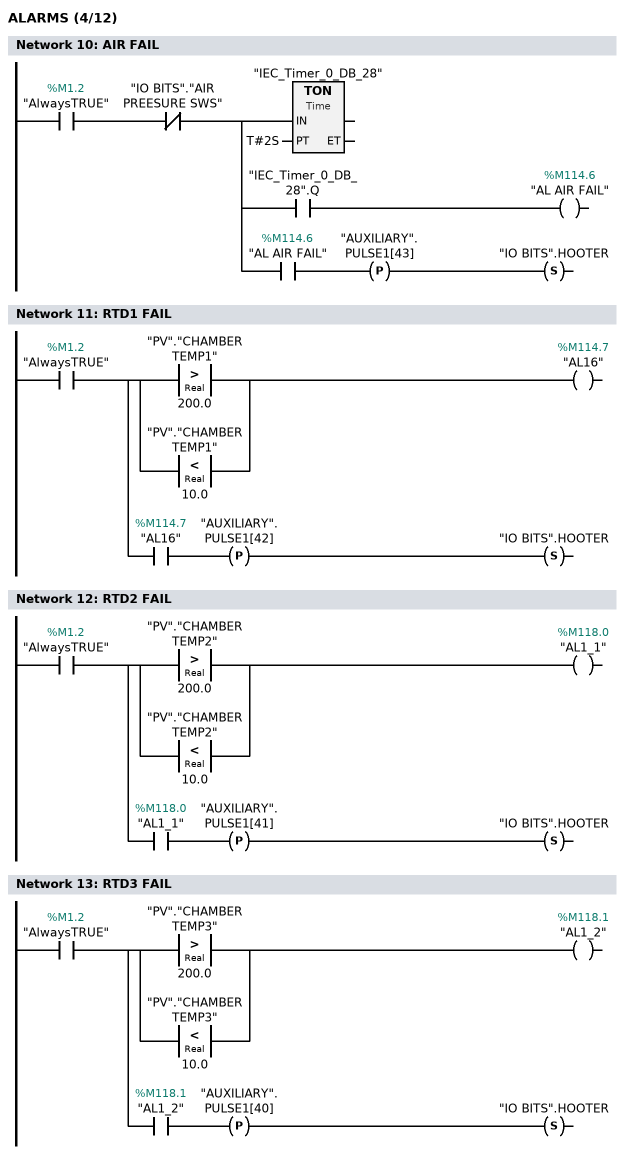
   RUNG wire#powerrail
      Contact( "AlwaysTRUE" )
      I_Contact( "IO BITS"."AIR PREESURE SWS" )
      wire#w1
      { S7_Templates := "time_type := Time" } "IEC_Timer_0_DB_28".TON(pt := T#2S, et =>)
   END_RUNG
   RUNG wire#w1
      Contact( "IEC_Timer_0_DB_28".Q )
      Coil( "AL AIR FAIL" )
   END_RUNG
   RUNG wire#w1
      Contact( "AL AIR FAIL" )
      P_Trig( "AUXILIARY".PULSE1[43] )
      S_Coil( "IO BITS".HOOTER )
   END_RUNG
   // the same network as SCL:
   #_w1 := "AlwaysTRUE" AND NOT "IO BITS"."AIR PREESURE SWS";
   "IEC_Timer_0_DB_28".TON(IN := #_w1, PT := T#2S);
   "AL AIR FAIL" := #_w1 AND "IEC_Timer_0_DB_28".Q;
   #_w2 := #_w1 AND "AL AIR FAIL";
   #_w3 := #_w2 AND NOT "AUXILIARY".PULSE1[43];   // rising edge
   "AUXILIARY".PULSE1[43] := #_w2;
   IF #_w3 THEN "IO BITS".HOOTER := TRUE; END_IF;
END_REGION

REGION Network 11: RTD1 FAIL
   RUNG wire#powerrail
      Contact( "AlwaysTRUE" )
      wire#w1
      { S7_Templates := "SrcType := Real" } GT_Contact(in1 := "PV"."CHAMBER TEMP1", in2 := 200.0)
      wire#w2
      Coil( "AL16" )
   END_RUNG
   RUNG wire#w1
      { S7_Templates := "SrcType := Real" } LT_Contact(in1 := "PV"."CHAMBER TEMP1", in2 := 10.0)
   END_RUNG wire#w2
   RUNG wire#w1
      Contact( "AL16" )
      P_Trig( "AUXILIARY".PULSE1[42] )
      S_Coil( "IO BITS".HOOTER )
   END_RUNG
   // the same network as SCL:
   "AL16" := "AlwaysTRUE" AND (("PV"."CHAMBER TEMP1" > 200.0) OR ("PV"."CHAMBER TEMP1" < 10.0));
   #_w1 := "AlwaysTRUE" AND "AL16";
   #_w2 := #_w1 AND NOT "AUXILIARY".PULSE1[42];   // rising edge
   "AUXILIARY".PULSE1[42] := #_w1;
   IF #_w2 THEN "IO BITS".HOOTER := TRUE; END_IF;
END_REGION

REGION Network 12: RTD2 FAIL
   RUNG wire#powerrail
      Contact( "AlwaysTRUE" )
      wire#w1
      { S7_Templates := "SrcType := Real" } GT_Contact(in1 := "PV"."CHAMBER TEMP2", in2 := 200.0)
      wire#w2
      Coil( "AL1_1" )
   END_RUNG
   RUNG wire#w1
      { S7_Templates := "SrcType := Real" } LT_Contact(in1 := "PV"."CHAMBER TEMP2", in2 := 10.0)
   END_RUNG wire#w2
   RUNG wire#w1
      Contact( "AL1_1" )
      P_Trig( "AUXILIARY".PULSE1[41] )
      S_Coil( "IO BITS".HOOTER )
   END_RUNG
   // the same network as SCL:
   "AL1_1" := "AlwaysTRUE" AND (("PV"."CHAMBER TEMP2" > 200.0) OR ("PV"."CHAMBER TEMP2" < 10.0));
   #_w1 := "AlwaysTRUE" AND "AL1_1";
   #_w2 := #_w1 AND NOT "AUXILIARY".PULSE1[41];   // rising edge
   "AUXILIARY".PULSE1[41] := #_w1;
   IF #_w2 THEN "IO BITS".HOOTER := TRUE; END_IF;
END_REGION

REGION Network 13: RTD3 FAIL
   RUNG wire#powerrail
      Contact( "AlwaysTRUE" )
      wire#w1
      { S7_Templates := "SrcType := Real" } GT_Contact(in1 := "PV"."CHAMBER TEMP3", in2 := 200.0)
      wire#w2
      Coil( "AL1_2" )
   END_RUNG
   RUNG wire#w1
      { S7_Templates := "SrcType := Real" } LT_Contact(in1 := "PV"."CHAMBER TEMP3", in2 := 10.0)
   END_RUNG wire#w2
   RUNG wire#w1
      Contact( "AL1_2" )
      P_Trig( "AUXILIARY".PULSE1[40] )
      S_Coil( "IO BITS".HOOTER )
   END_RUNG
   // the same network as SCL:
   "AL1_2" := "AlwaysTRUE" AND (("PV"."CHAMBER TEMP3" > 200.0) OR ("PV"."CHAMBER TEMP3" < 10.0));
   #_w1 := "AlwaysTRUE" AND "AL1_2";
   #_w2 := #_w1 AND NOT "AUXILIARY".PULSE1[40];   // rising edge
   "AUXILIARY".PULSE1[40] := #_w1;
   IF #_w2 THEN "IO BITS".HOOTER := TRUE; END_IF;
END_REGION

REGION Network 14: RTD4 FAIL
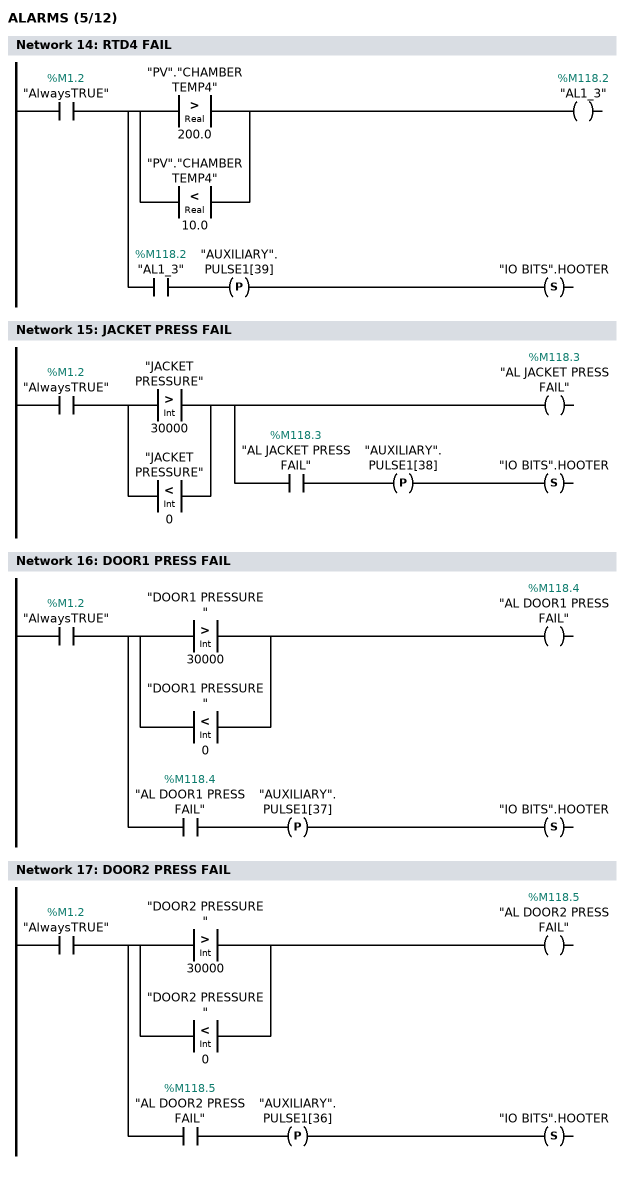
   RUNG wire#powerrail
      Contact( "AlwaysTRUE" )
      wire#w1
      { S7_Templates := "SrcType := Real" } GT_Contact(in1 := "PV"."CHAMBER TEMP4", in2 := 200.0)
      wire#w2
      Coil( "AL1_3" )
   END_RUNG
   RUNG wire#w1
      { S7_Templates := "SrcType := Real" } LT_Contact(in1 := "PV"."CHAMBER TEMP4", in2 := 10.0)
   END_RUNG wire#w2
   RUNG wire#w1
      Contact( "AL1_3" )
      P_Trig( "AUXILIARY".PULSE1[39] )
      S_Coil( "IO BITS".HOOTER )
   END_RUNG
   // the same network as SCL:
   "AL1_3" := "AlwaysTRUE" AND (("PV"."CHAMBER TEMP4" > 200.0) OR ("PV"."CHAMBER TEMP4" < 10.0));
   #_w1 := "AlwaysTRUE" AND "AL1_3";
   #_w2 := #_w1 AND NOT "AUXILIARY".PULSE1[39];   // rising edge
   "AUXILIARY".PULSE1[39] := #_w1;
   IF #_w2 THEN "IO BITS".HOOTER := TRUE; END_IF;
END_REGION

REGION Network 15: JACKET PRESS FAIL
   RUNG wire#powerrail
      Contact( "AlwaysTRUE" )
      wire#w1
      { S7_Templates := "SrcType := Int" } GT_Contact(in1 := "JACKET PRESSURE", in2 := 30000)
      wire#w2
      Coil( "AL JACKET PRESS FAIL" )
   END_RUNG
   RUNG wire#w1
      { S7_Templates := "SrcType := Int" } LT_Contact(in1 := "JACKET PRESSURE", in2 := 0)
   END_RUNG wire#w2
   RUNG wire#w2
      Contact( "AL JACKET PRESS FAIL" )
      P_Trig( "AUXILIARY".PULSE1[38] )
      S_Coil( "IO BITS".HOOTER )
   END_RUNG
   // the same network as SCL:
   "AL JACKET PRESS FAIL" := "AlwaysTRUE" AND (("JACKET PRESSURE" > 30000) OR ("JACKET PRESSURE" < 0));
   #_w1 := "AL JACKET PRESS FAIL" AND "AL JACKET PRESS FAIL";
   #_w2 := #_w1 AND NOT "AUXILIARY".PULSE1[38];   // rising edge
   "AUXILIARY".PULSE1[38] := #_w1;
   IF #_w2 THEN "IO BITS".HOOTER := TRUE; END_IF;
END_REGION

REGION Network 16: DOOR1 PRESS FAIL
   RUNG wire#powerrail
      Contact( "AlwaysTRUE" )
      wire#w1
      { S7_Templates := "SrcType := Int" } GT_Contact(in1 := "DOOR1 PRESSURE", in2 := 30000)
      wire#w2
      Coil( "AL DOOR1 PRESS FAIL" )
   END_RUNG
   RUNG wire#w1
      { S7_Templates := "SrcType := Int" } LT_Contact(in1 := "DOOR1 PRESSURE", in2 := 0)
   END_RUNG wire#w2
   RUNG wire#w1
      Contact( "AL DOOR1 PRESS FAIL" )
      P_Trig( "AUXILIARY".PULSE1[37] )
      S_Coil( "IO BITS".HOOTER )
   END_RUNG
   // the same network as SCL:
   "AL DOOR1 PRESS FAIL" := "AlwaysTRUE" AND (("DOOR1 PRESSURE" > 30000) OR ("DOOR1 PRESSURE" < 0));
   #_w1 := "AlwaysTRUE" AND "AL DOOR1 PRESS FAIL";
   #_w2 := #_w1 AND NOT "AUXILIARY".PULSE1[37];   // rising edge
   "AUXILIARY".PULSE1[37] := #_w1;
   IF #_w2 THEN "IO BITS".HOOTER := TRUE; END_IF;
END_REGION

REGION Network 17: DOOR2 PRESS FAIL
   RUNG wire#powerrail
      Contact( "AlwaysTRUE" )
      wire#w1
      { S7_Templates := "SrcType := Int" } GT_Contact(in1 := "DOOR2 PRESSURE", in2 := 30000)
      wire#w2
      Coil( "AL DOOR2 PRESS FAIL" )
   END_RUNG
   RUNG wire#w1
      { S7_Templates := "SrcType := Int" } LT_Contact(in1 := "DOOR2 PRESSURE", in2 := 0)
   END_RUNG wire#w2
   RUNG wire#w1
      Contact( "AL DOOR2 PRESS FAIL" )
      P_Trig( "AUXILIARY".PULSE1[36] )
      S_Coil( "IO BITS".HOOTER )
   END_RUNG
   // the same network as SCL:
   "AL DOOR2 PRESS FAIL" := "AlwaysTRUE" AND (("DOOR2 PRESSURE" > 30000) OR ("DOOR2 PRESSURE" < 0));
   #_w1 := "AlwaysTRUE" AND "AL DOOR2 PRESS FAIL";
   #_w2 := #_w1 AND NOT "AUXILIARY".PULSE1[36];   // rising edge
   "AUXILIARY".PULSE1[36] := #_w1;
   IF #_w2 THEN "IO BITS".HOOTER := TRUE; END_IF;
END_REGION

REGION Network 18: chamber press fail
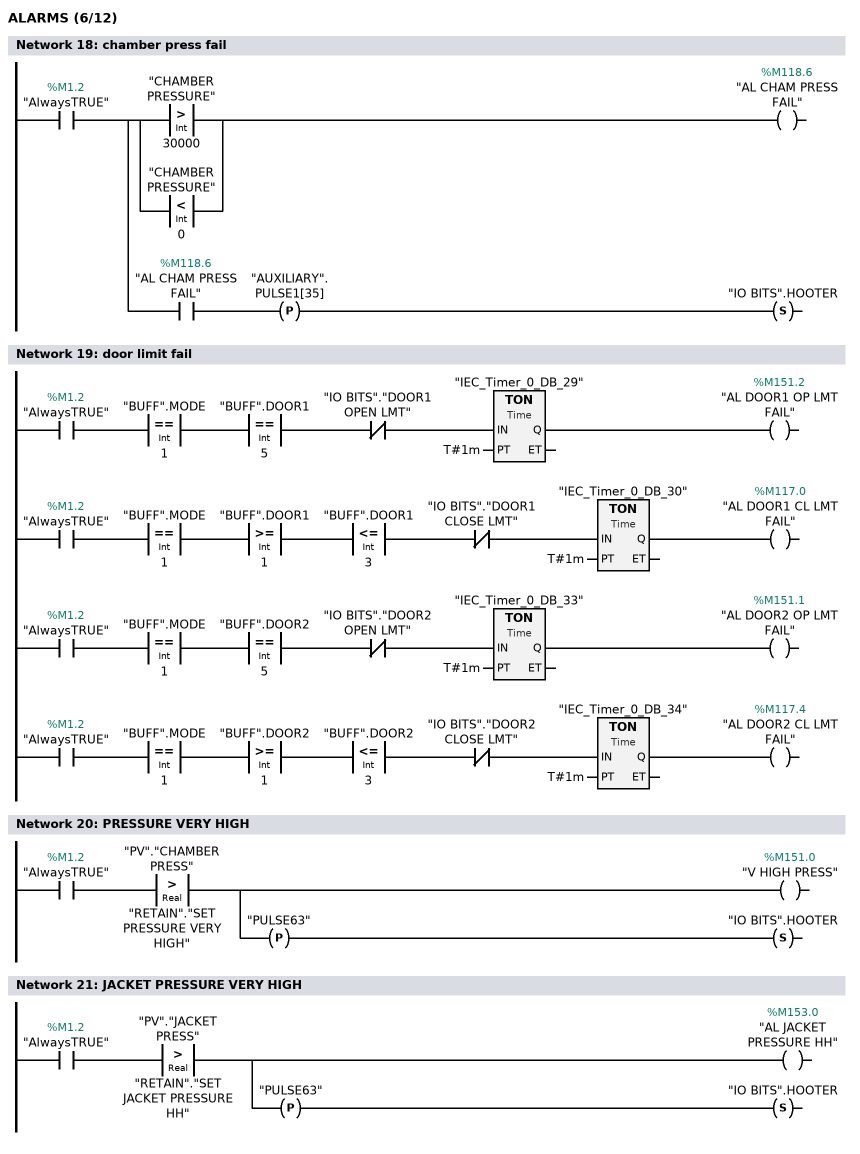
   RUNG wire#powerrail
      Contact( "AlwaysTRUE" )
      wire#w1
      { S7_Templates := "SrcType := Int" } GT_Contact(in1 := "CHAMBER PRESSURE", in2 := 30000)
      wire#w2
      Coil( "AL CHAM PRESS FAIL" )
   END_RUNG
   RUNG wire#w1
      { S7_Templates := "SrcType := Int" } LT_Contact(in1 := "CHAMBER PRESSURE", in2 := 0)
   END_RUNG wire#w2
   RUNG wire#w1
      Contact( "AL CHAM PRESS FAIL" )
      P_Trig( "AUXILIARY".PULSE1[35] )
      S_Coil( "IO BITS".HOOTER )
   END_RUNG
   // the same network as SCL:
   "AL CHAM PRESS FAIL" := "AlwaysTRUE" AND (("CHAMBER PRESSURE" > 30000) OR ("CHAMBER PRESSURE" < 0));
   #_w1 := "AlwaysTRUE" AND "AL CHAM PRESS FAIL";
   #_w2 := #_w1 AND NOT "AUXILIARY".PULSE1[35];   // rising edge
   "AUXILIARY".PULSE1[35] := #_w1;
   IF #_w2 THEN "IO BITS".HOOTER := TRUE; END_IF;
END_REGION

REGION Network 19: door limit fail
   RUNG wire#powerrail
      Contact( "AlwaysTRUE" )
      { S7_Templates := "SrcType := Int" } EQ_Contact(in1 := "BUFF".MODE, in2 := 1)
      { S7_Templates := "SrcType := Int" } EQ_Contact(in1 := "BUFF".DOOR1, in2 := 5)
      I_Contact( "IO BITS"."DOOR1 OPEN LMT" )
      { S7_Templates := "time_type := Time" } "IEC_Timer_0_DB_29".TON(pt := T#1m, et =>)
      Coil( "AL DOOR1 OP LMT FAIL" )
   END_RUNG
   RUNG wire#powerrail
      Contact( "AlwaysTRUE" )
      { S7_Templates := "SrcType := Int" } EQ_Contact(in1 := "BUFF".MODE, in2 := 1)
      { S7_Templates := "SrcType := Int" } GE_Contact(in1 := "BUFF".DOOR1, in2 := 1)
      { S7_Templates := "SrcType := Int" } LE_Contact(in1 := "BUFF".DOOR1, in2 := 3)
      I_Contact( "IO BITS"."DOOR1 CLOSE LMT" )
      { S7_Templates := "time_type := Time" } "IEC_Timer_0_DB_30".TON(pt := T#1m, et =>)
      Coil( "AL DOOR1 CL LMT FAIL" )
   END_RUNG
   RUNG wire#powerrail
      Contact( "AlwaysTRUE" )
      { S7_Templates := "SrcType := Int" } EQ_Contact(in1 := "BUFF".MODE, in2 := 1)
      { S7_Templates := "SrcType := Int" } EQ_Contact(in1 := "BUFF".DOOR2, in2 := 5)
      I_Contact( "IO BITS"."DOOR2 OPEN LMT" )
      { S7_Templates := "time_type := Time" } "IEC_Timer_0_DB_33".TON(pt := T#1m, et =>)
      Coil( "AL DOOR2 OP LMT FAIL" )
   END_RUNG
   RUNG wire#powerrail
      Contact( "AlwaysTRUE" )
      { S7_Templates := "SrcType := Int" } EQ_Contact(in1 := "BUFF".MODE, in2 := 1)
      { S7_Templates := "SrcType := Int" } GE_Contact(in1 := "BUFF".DOOR2, in2 := 1)
      { S7_Templates := "SrcType := Int" } LE_Contact(in1 := "BUFF".DOOR2, in2 := 3)
      I_Contact( "IO BITS"."DOOR2 CLOSE LMT" )
      { S7_Templates := "time_type := Time" } "IEC_Timer_0_DB_34".TON(pt := T#1m, et =>)
      Coil( "AL DOOR2 CL LMT FAIL" )
   END_RUNG
   // the same network as SCL:
   "IEC_Timer_0_DB_29".TON(IN := "AlwaysTRUE" AND ("BUFF".MODE = 1) AND ("BUFF".DOOR1 = 5) AND NOT "IO BITS"."DOOR1 OPEN LMT",
                           PT := T#1m);
   "AL DOOR1 OP LMT FAIL" := "IEC_Timer_0_DB_29".Q;
   "IEC_Timer_0_DB_30".TON(IN := "AlwaysTRUE" AND ("BUFF".MODE = 1) AND ("BUFF".DOOR1 >= 1) AND ("BUFF".DOOR1 <= 3) AND NOT "IO BITS"."DOOR1 CLOSE LMT",
                           PT := T#1m);
   "AL DOOR1 CL LMT FAIL" := "IEC_Timer_0_DB_30".Q;
   "IEC_Timer_0_DB_33".TON(IN := "AlwaysTRUE" AND ("BUFF".MODE = 1) AND ("BUFF".DOOR2 = 5) AND NOT "IO BITS"."DOOR2 OPEN LMT",
                           PT := T#1m);
   "AL DOOR2 OP LMT FAIL" := "IEC_Timer_0_DB_33".Q;
   "IEC_Timer_0_DB_34".TON(IN := "AlwaysTRUE" AND ("BUFF".MODE = 1) AND ("BUFF".DOOR2 >= 1) AND ("BUFF".DOOR2 <= 3) AND NOT "IO BITS"."DOOR2 CLOSE LMT",
                           PT := T#1m);
   "AL DOOR2 CL LMT FAIL" := "IEC_Timer_0_DB_34".Q;
END_REGION

REGION Network 20: PRESSURE VERY HIGH
   RUNG wire#powerrail
      Contact( "AlwaysTRUE" )
      { S7_Templates := "SrcType := Real" } GT_Contact(in1 := "PV"."CHAMBER PRESS", in2 := "RETAIN"."SET PRESSURE VERY HIGH")
      wire#w1
      Coil( "V HIGH PRESS" )
   END_RUNG
   RUNG wire#w1
      P_Trig( "PULSE63" )
      S_Coil( "IO BITS".HOOTER )
   END_RUNG
   // the same network as SCL:
   "V HIGH PRESS" := "AlwaysTRUE" AND ("PV"."CHAMBER PRESS" > "RETAIN"."SET PRESSURE VERY HIGH");
   #_w1 := "V HIGH PRESS" AND NOT "PULSE63";   // rising edge
   "PULSE63" := "V HIGH PRESS";
   IF #_w1 THEN "IO BITS".HOOTER := TRUE; END_IF;
END_REGION

REGION Network 21: JACKET PRESSURE VERY HIGH
   RUNG wire#powerrail
      Contact( "AlwaysTRUE" )
      { S7_Templates := "SrcType := Real" } GT_Contact(in1 := "PV"."JACKET PRESS", in2 := "RETAIN"."SET JACKET PRESSURE HH")
      wire#w1
      Coil( "AL JACKET PRESSURE HH" )
   END_RUNG
   RUNG wire#w1
      P_Trig( "PULSE63" )
      S_Coil( "IO BITS".HOOTER )
   END_RUNG
   // the same network as SCL:
   "AL JACKET PRESSURE HH" := "AlwaysTRUE" AND ("PV"."JACKET PRESS" > "RETAIN"."SET JACKET PRESSURE HH");
   #_w1 := "AL JACKET PRESSURE HH" AND NOT "PULSE63";   // rising edge
   "PULSE63" := "AL JACKET PRESSURE HH";
   IF #_w1 THEN "IO BITS".HOOTER := TRUE; END_IF;
END_REGION

REGION Network 22: TEMPERATURE OVERSHOOT
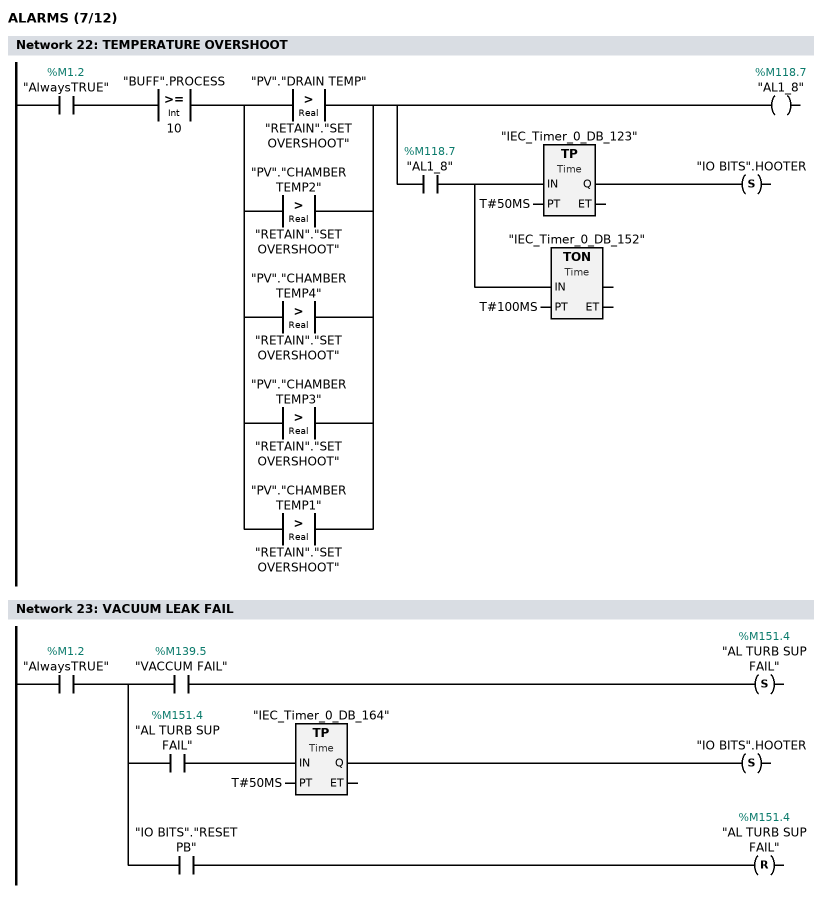
   RUNG wire#powerrail
      Contact( "AlwaysTRUE" )
      { S7_Templates := "SrcType := Int" } GE_Contact(in1 := "BUFF".PROCESS, in2 := 10)
      wire#w1
      { S7_Templates := "SrcType := Real" } GT_Contact(in1 := "PV"."DRAIN TEMP", in2 := "RETAIN"."SET OVERSHOOT")
      wire#w2
      Coil( "AL1_8" )
   END_RUNG
   RUNG wire#w1
      { S7_Templates := "SrcType := Real" } GT_Contact(in1 := "PV"."CHAMBER TEMP2", in2 := "RETAIN"."SET OVERSHOOT")
   END_RUNG wire#w2
   RUNG wire#w1
      { S7_Templates := "SrcType := Real" } GT_Contact(in1 := "PV"."CHAMBER TEMP4", in2 := "RETAIN"."SET OVERSHOOT")
   END_RUNG wire#w2
   RUNG wire#w1
      { S7_Templates := "SrcType := Real" } GT_Contact(in1 := "PV"."CHAMBER TEMP3", in2 := "RETAIN"."SET OVERSHOOT")
   END_RUNG wire#w2
   RUNG wire#w1
      { S7_Templates := "SrcType := Real" } GT_Contact(in1 := "PV"."CHAMBER TEMP1", in2 := "RETAIN"."SET OVERSHOOT")
   END_RUNG wire#w2
   RUNG wire#w2
      Contact( "AL1_8" )
      wire#w3
      { S7_Templates := "time_type := Time" } "IEC_Timer_0_DB_123".TP(pt := T#50MS, et =>)
      S_Coil( "IO BITS".HOOTER )
   END_RUNG
   RUNG wire#w3
      { S7_Templates := "time_type := Time" } "IEC_Timer_0_DB_152".TON(pt := T#100MS, et =>)
   END_RUNG
   // the same network as SCL:
   "AL1_8" := "AlwaysTRUE" AND ("BUFF".PROCESS >= 10) AND (("PV"."DRAIN TEMP" > "RETAIN"."SET OVERSHOOT") OR ("PV"."CHAMBER TEMP2" > "RETAIN"."SET OVERSHOOT") OR ("PV"."CHAMBER TEMP4" > "RETAIN"."SET OVERSHOOT") OR ("PV"."CHAMBER TEMP3" > "RETAIN"."SET OVERSHOOT") OR ("PV"."CHAMBER TEMP1" > "RETAIN"."SET OVERSHOOT"));
   #_w1 := "AL1_8" AND "AL1_8";
   "IEC_Timer_0_DB_123".TP(IN := #_w1, PT := T#50MS);
   IF "IEC_Timer_0_DB_123".Q THEN "IO BITS".HOOTER := TRUE; END_IF;
   "IEC_Timer_0_DB_152".TON(IN := #_w1, PT := T#100MS);
END_REGION

REGION Network 23: VACUUM LEAK FAIL
   RUNG wire#powerrail
      Contact( "AlwaysTRUE" )
      wire#w1
      Contact( "VACCUM FAIL" )
      S_Coil( "AL TURB SUP FAIL" )
   END_RUNG
   RUNG wire#w1
      Contact( "AL TURB SUP FAIL" )
      { S7_Templates := "time_type := Time" } "IEC_Timer_0_DB_164".TP(pt := T#50MS, et =>)
      S_Coil( "IO BITS".HOOTER )
   END_RUNG
   RUNG wire#w1
      Contact( "IO BITS"."RESET PB" )
      R_Coil( "AL TURB SUP FAIL" )
   END_RUNG
   // the same network as SCL:
   IF "AlwaysTRUE" AND "VACCUM FAIL" THEN "AL TURB SUP FAIL" := TRUE; END_IF;
   "IEC_Timer_0_DB_164".TP(IN := "AlwaysTRUE" AND "AL TURB SUP FAIL", PT := T#50MS);
   IF "IEC_Timer_0_DB_164".Q THEN "IO BITS".HOOTER := TRUE; END_IF;
   IF "AlwaysTRUE" AND "IO BITS"."RESET PB" THEN "AL TURB SUP FAIL" := FALSE; END_IF;
END_REGION

REGION Network 24: vacuum break fail
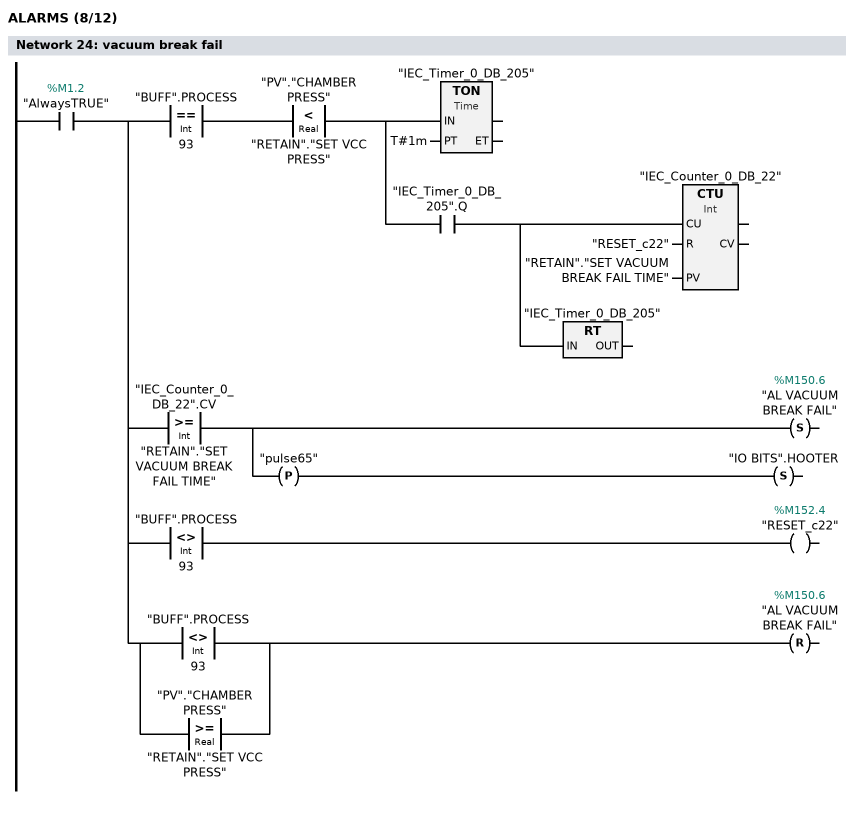
   RUNG wire#powerrail
      Contact( "AlwaysTRUE" )
      wire#w1
      { S7_Templates := "SrcType := Int" } EQ_Contact(in1 := "BUFF".PROCESS, in2 := 93)
      { S7_Templates := "SrcType := Real" } LT_Contact(in1 := "PV"."CHAMBER PRESS", in2 := "RETAIN"."SET VCC PRESS")
      wire#w2
      { S7_Templates := "time_type := Time" } "IEC_Timer_0_DB_205".TON(pt := T#1m, et =>)
   END_RUNG
   RUNG wire#w2
      Contact( "IEC_Timer_0_DB_205".Q )
      wire#w3
      { S7_Templates := "value_type := Int" } "IEC_Counter_0_DB_22".CTU(r := "RESET_c22", pv := "RETAIN"."SET VACUUM BREAK FAIL TIME", cv =>)
   END_RUNG
   RUNG wire#w3
      RT_Coil( "IEC_Timer_0_DB_205" )
   END_RUNG
   RUNG wire#w1
      { S7_Templates := "SrcType := Int" } GE_Contact(in1 := "IEC_Counter_0_DB_22".CV, in2 := "RETAIN"."SET VACUUM BREAK FAIL TIME")
      wire#w4
      S_Coil( "AL VACUUM BREAK FAIL" )
   END_RUNG
   RUNG wire#w4
      P_Trig( "pulse65" )
      S_Coil( "IO BITS".HOOTER )
   END_RUNG
   RUNG wire#w1
      { S7_Templates := "SrcType := Int" } NE_Contact(in1 := "BUFF".PROCESS, in2 := 93)
      Coil( "RESET_c22" )
   END_RUNG
   RUNG wire#w1
      { S7_Templates := "SrcType := Int" } NE_Contact(in1 := "BUFF".PROCESS, in2 := 93)
      wire#w5
      R_Coil( "AL VACUUM BREAK FAIL" )
   END_RUNG
   RUNG wire#w1
      { S7_Templates := "SrcType := Real" } GE_Contact(in1 := "PV"."CHAMBER PRESS", in2 := "RETAIN"."SET VCC PRESS")
   END_RUNG wire#w5
   // the same network as SCL:
   #_w1 := "AlwaysTRUE" AND ("BUFF".PROCESS = 93) AND ("PV"."CHAMBER PRESS" < "RETAIN"."SET VCC PRESS");
   "IEC_Timer_0_DB_205".TON(IN := #_w1, PT := T#1m);
   #_w2 := #_w1 AND "IEC_Timer_0_DB_205".Q;
   "IEC_Counter_0_DB_22".CTU(CU := #_w2, R := "RESET_c22", PV := "RETAIN"."SET VACUUM BREAK FAIL TIME");
   IF #_w2 THEN RESET_TIMER("IEC_Timer_0_DB_205"); END_IF;
   #_w3 := "AlwaysTRUE" AND ("IEC_Counter_0_DB_22".CV >= "RETAIN"."SET VACUUM BREAK FAIL TIME");
   IF #_w3 THEN "AL VACUUM BREAK FAIL" := TRUE; END_IF;
   #_w4 := #_w3 AND NOT "pulse65";   // rising edge
   "pulse65" := #_w3;
   IF #_w4 THEN "IO BITS".HOOTER := TRUE; END_IF;
   "RESET_c22" := "AlwaysTRUE" AND ("BUFF".PROCESS <> 93);
   IF "AlwaysTRUE" AND (("BUFF".PROCESS <> 93) OR ("PV"."CHAMBER PRESS" >= "RETAIN"."SET VCC PRESS")) THEN
       "AL VACUUM BREAK FAIL" := FALSE;
   END_IF;
END_REGION

REGION Network 25: JACKET ALARM TIME
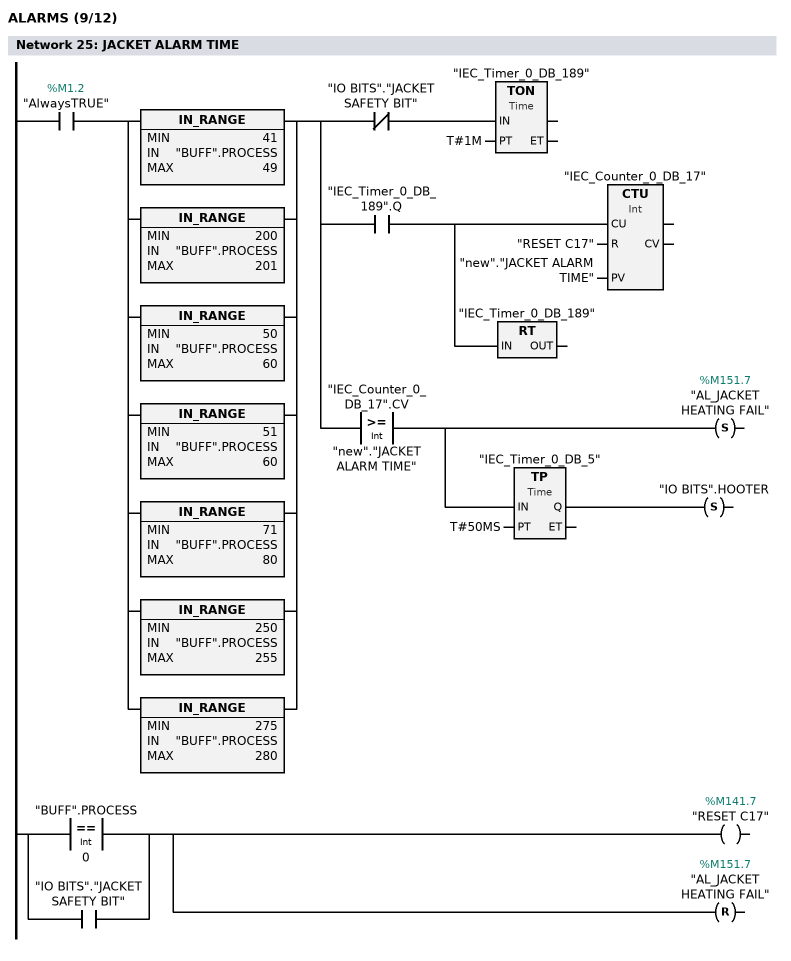
   RUNG wire#powerrail
      Contact( "AlwaysTRUE" )
      wire#w1
      { S7_Templates := "SrcType := Int" } InRange(min := 41, in := "BUFF".PROCESS, max := 49)
      wire#w2
      I_Contact( "IO BITS"."JACKET SAFETY BIT" )
      { S7_Templates := "time_type := Time" } "IEC_Timer_0_DB_189".TON(pt := T#1M, et =>)
   END_RUNG
   RUNG wire#w1
      { S7_Templates := "SrcType := Int" } InRange(min := 200, in := "BUFF".PROCESS, max := 201)
   END_RUNG wire#w2
   RUNG wire#w1
      { S7_Templates := "SrcType := Int" } InRange(min := 50, in := "BUFF".PROCESS, max := 60)
   END_RUNG wire#w2
   RUNG wire#w1
      { S7_Templates := "SrcType := Int" } InRange(min := 51, in := "BUFF".PROCESS, max := 60)
   END_RUNG wire#w2
   RUNG wire#w1
      { S7_Templates := "SrcType := Int" } InRange(min := 71, in := "BUFF".PROCESS, max := 80)
   END_RUNG wire#w2
   RUNG wire#w1
      { S7_Templates := "SrcType := Int" } InRange(min := 250, in := "BUFF".PROCESS, max := 255)
   END_RUNG wire#w2
   RUNG wire#w1
      { S7_Templates := "SrcType := Int" } InRange(min := 275, in := "BUFF".PROCESS, max := 280)
   END_RUNG wire#w2
   RUNG wire#w2
      Contact( "IEC_Timer_0_DB_189".Q )
      wire#w3
      { S7_Templates := "value_type := Int" } "IEC_Counter_0_DB_17".CTU(r := "RESET C17", pv := "new"."JACKET ALARM TIME", cv =>)
   END_RUNG
   RUNG wire#w3
      RT_Coil( "IEC_Timer_0_DB_189" )
   END_RUNG
   RUNG wire#w2
      { S7_Templates := "SrcType := Int" } GE_Contact(in1 := "IEC_Counter_0_DB_17".CV, in2 := "new"."JACKET ALARM TIME")
      wire#w4
      S_Coil( "AL_JACKET HEATING FAIL" )
   END_RUNG
   RUNG wire#w4
      { S7_Templates := "time_type := Time" } "IEC_Timer_0_DB_5".TP(pt := T#50MS, et =>)
      S_Coil( "IO BITS".HOOTER )
   END_RUNG
   RUNG wire#powerrail
      { S7_Templates := "SrcType := Int" } EQ_Contact(in1 := "BUFF".PROCESS, in2 := 0)
      wire#w5
      Coil( "RESET C17" )
   END_RUNG
   RUNG wire#powerrail
      Contact( "IO BITS"."JACKET SAFETY BIT" )
   END_RUNG wire#w5
   RUNG wire#w5
      R_Coil( "AL_JACKET HEATING FAIL" )
   END_RUNG
   // the same network as SCL:
   #_w1 := "AlwaysTRUE" AND (((41 <= "BUFF".PROCESS) AND ("BUFF".PROCESS <= 49)) OR ((200 <= "BUFF".PROCESS) AND ("BUFF".PROCESS <= 201)) OR ((50 <= "BUFF".PROCESS) AND ("BUFF".PROCESS <= 60)) OR ((51 <= "BUFF".PROCESS) AND ("BUFF".PROCESS <= 60)) OR ((71 <= "BUFF".PROCESS) AND ("BUFF".PROCESS <= 80)) OR ((250 <= "BUFF".PROCESS) AND ("BUFF".PROCESS <= 255)) OR ((275 <= "BUFF".PROCESS) AND ("BUFF".PROCESS <= 280)));
   "IEC_Timer_0_DB_189".TON(IN := #_w1 AND NOT "IO BITS"."JACKET SAFETY BIT", PT := T#1M);
   #_w2 := #_w1 AND "IEC_Timer_0_DB_189".Q;
   "IEC_Counter_0_DB_17".CTU(CU := #_w2, R := "RESET C17", PV := "new"."JACKET ALARM TIME");
   IF #_w2 THEN RESET_TIMER("IEC_Timer_0_DB_189"); END_IF;
   #_w3 := #_w1 AND ("IEC_Counter_0_DB_17".CV >= "new"."JACKET ALARM TIME");
   IF #_w3 THEN "AL_JACKET HEATING FAIL" := TRUE; END_IF;
   "IEC_Timer_0_DB_5".TP(IN := #_w3, PT := T#50MS);
   IF "IEC_Timer_0_DB_5".Q THEN "IO BITS".HOOTER := TRUE; END_IF;
   "RESET C17" := ("BUFF".PROCESS = 0) OR "IO BITS"."JACKET SAFETY BIT";
   IF "RESET C17" THEN "AL_JACKET HEATING FAIL" := FALSE; END_IF;
END_REGION

REGION Network 26: heatup ALARM TIME
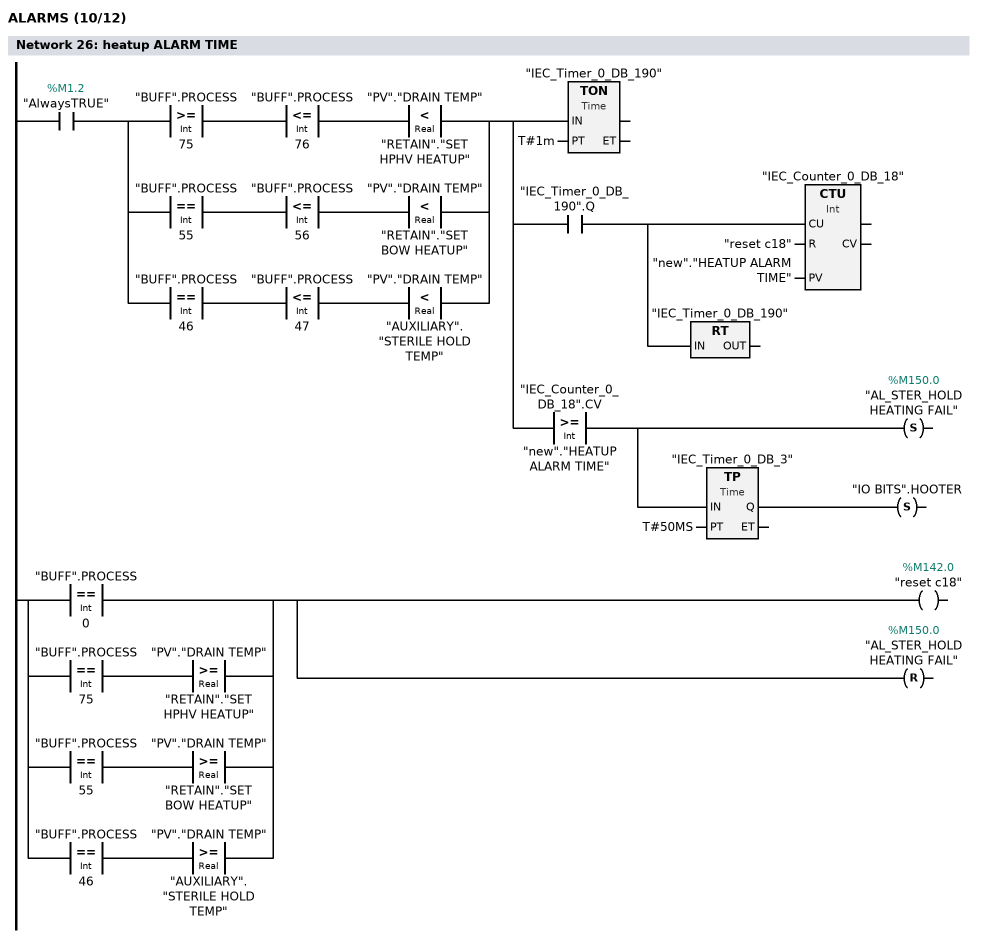
   RUNG wire#powerrail
      Contact( "AlwaysTRUE" )
      wire#w1
      { S7_Templates := "SrcType := Int" } GE_Contact(in1 := "BUFF".PROCESS, in2 := 75)
      { S7_Templates := "SrcType := Int" } LE_Contact(in1 := "BUFF".PROCESS, in2 := 76)
      { S7_Templates := "SrcType := Real" } LT_Contact(in1 := "PV"."DRAIN TEMP", in2 := "RETAIN"."SET HPHV HEATUP")
      wire#w2
      { S7_Templates := "time_type := Time" } "IEC_Timer_0_DB_190".TON(pt := T#1m, et =>)
   END_RUNG
   RUNG wire#w1
      { S7_Templates := "SrcType := Int" } EQ_Contact(in1 := "BUFF".PROCESS, in2 := 55)
      { S7_Templates := "SrcType := Int" } LE_Contact(in1 := "BUFF".PROCESS, in2 := 56)
      { S7_Templates := "SrcType := Real" } LT_Contact(in1 := "PV"."DRAIN TEMP", in2 := "RETAIN"."SET BOW HEATUP")
   END_RUNG wire#w2
   RUNG wire#w1
      { S7_Templates := "SrcType := Int" } EQ_Contact(in1 := "BUFF".PROCESS, in2 := 46)
      { S7_Templates := "SrcType := Int" } LE_Contact(in1 := "BUFF".PROCESS, in2 := 47)
      { S7_Templates := "SrcType := Real" } LT_Contact(in1 := "PV"."DRAIN TEMP", in2 := "AUXILIARY"."STERILE HOLD TEMP")
   END_RUNG wire#w2
   RUNG wire#w2
      Contact( "IEC_Timer_0_DB_190".Q )
      wire#w3
      { S7_Templates := "value_type := Int" } "IEC_Counter_0_DB_18".CTU(r := "reset c18", pv := "new"."HEATUP ALARM TIME", cv =>)
   END_RUNG
   RUNG wire#w3
      RT_Coil( "IEC_Timer_0_DB_190" )
   END_RUNG
   RUNG wire#w2
      { S7_Templates := "SrcType := Int" } GE_Contact(in1 := "IEC_Counter_0_DB_18".CV, in2 := "new"."HEATUP ALARM TIME")
      wire#w4
      S_Coil( "AL_STER_HOLD HEATING FAIL" )
   END_RUNG
   RUNG wire#w4
      { S7_Templates := "time_type := Time" } "IEC_Timer_0_DB_3".TP(pt := T#50MS, et =>)
      S_Coil( "IO BITS".HOOTER )
   END_RUNG
   RUNG wire#powerrail
      { S7_Templates := "SrcType := Int" } EQ_Contact(in1 := "BUFF".PROCESS, in2 := 0)
      wire#w5
      Coil( "reset c18" )
   END_RUNG
   RUNG wire#powerrail
      { S7_Templates := "SrcType := Int" } EQ_Contact(in1 := "BUFF".PROCESS, in2 := 75)
      { S7_Templates := "SrcType := Real" } GE_Contact(in1 := "PV"."DRAIN TEMP", in2 := "RETAIN"."SET HPHV HEATUP")
   END_RUNG wire#w5
   RUNG wire#powerrail
      { S7_Templates := "SrcType := Int" } EQ_Contact(in1 := "BUFF".PROCESS, in2 := 55)
      { S7_Templates := "SrcType := Real" } GE_Contact(in1 := "PV"."DRAIN TEMP", in2 := "RETAIN"."SET BOW HEATUP")
   END_RUNG wire#w5
   RUNG wire#powerrail
      { S7_Templates := "SrcType := Int" } EQ_Contact(in1 := "BUFF".PROCESS, in2 := 46)
      { S7_Templates := "SrcType := Real" } GE_Contact(in1 := "PV"."DRAIN TEMP", in2 := "AUXILIARY"."STERILE HOLD TEMP")
   END_RUNG wire#w5
   RUNG wire#w5
      R_Coil( "AL_STER_HOLD HEATING FAIL" )
   END_RUNG
   // the same network as SCL:
   #_w1 := "AlwaysTRUE" AND ((("BUFF".PROCESS >= 75) AND ("BUFF".PROCESS <= 76) AND ("PV"."DRAIN TEMP" < "RETAIN"."SET HPHV HEATUP")) OR (("BUFF".PROCESS = 55) AND ("BUFF".PROCESS <= 56) AND ("PV"."DRAIN TEMP" < "RETAIN"."SET BOW HEATUP")) OR (("BUFF".PROCESS = 46) AND ("BUFF".PROCESS <= 47) AND ("PV"."DRAIN TEMP" < "AUXILIARY"."STERILE HOLD TEMP")));
   "IEC_Timer_0_DB_190".TON(IN := #_w1, PT := T#1m);
   #_w2 := #_w1 AND "IEC_Timer_0_DB_190".Q;
   "IEC_Counter_0_DB_18".CTU(CU := #_w2, R := "reset c18", PV := "new"."HEATUP ALARM TIME");
   IF #_w2 THEN RESET_TIMER("IEC_Timer_0_DB_190"); END_IF;
   #_w3 := #_w1 AND ("IEC_Counter_0_DB_18".CV >= "new"."HEATUP ALARM TIME");
   IF #_w3 THEN "AL_STER_HOLD HEATING FAIL" := TRUE; END_IF;
   "IEC_Timer_0_DB_3".TP(IN := #_w3, PT := T#50MS);
   IF "IEC_Timer_0_DB_3".Q THEN "IO BITS".HOOTER := TRUE; END_IF;
   "reset c18" := ("BUFF".PROCESS = 0) OR (("BUFF".PROCESS = 75) AND ("PV"."DRAIN TEMP" >= "RETAIN"."SET HPHV HEATUP")) OR (("BUFF".PROCESS = 55) AND ("PV"."DRAIN TEMP" >= "RETAIN"."SET BOW HEATUP")) OR (("BUFF".PROCESS = 46) AND ("PV"."DRAIN TEMP" >= "AUXILIARY"."STERILE HOLD TEMP"));
   IF "reset c18" THEN "AL_STER_HOLD HEATING FAIL" := FALSE; END_IF;
END_REGION

REGION Network 27: VACUUM NOT AVAILABLE
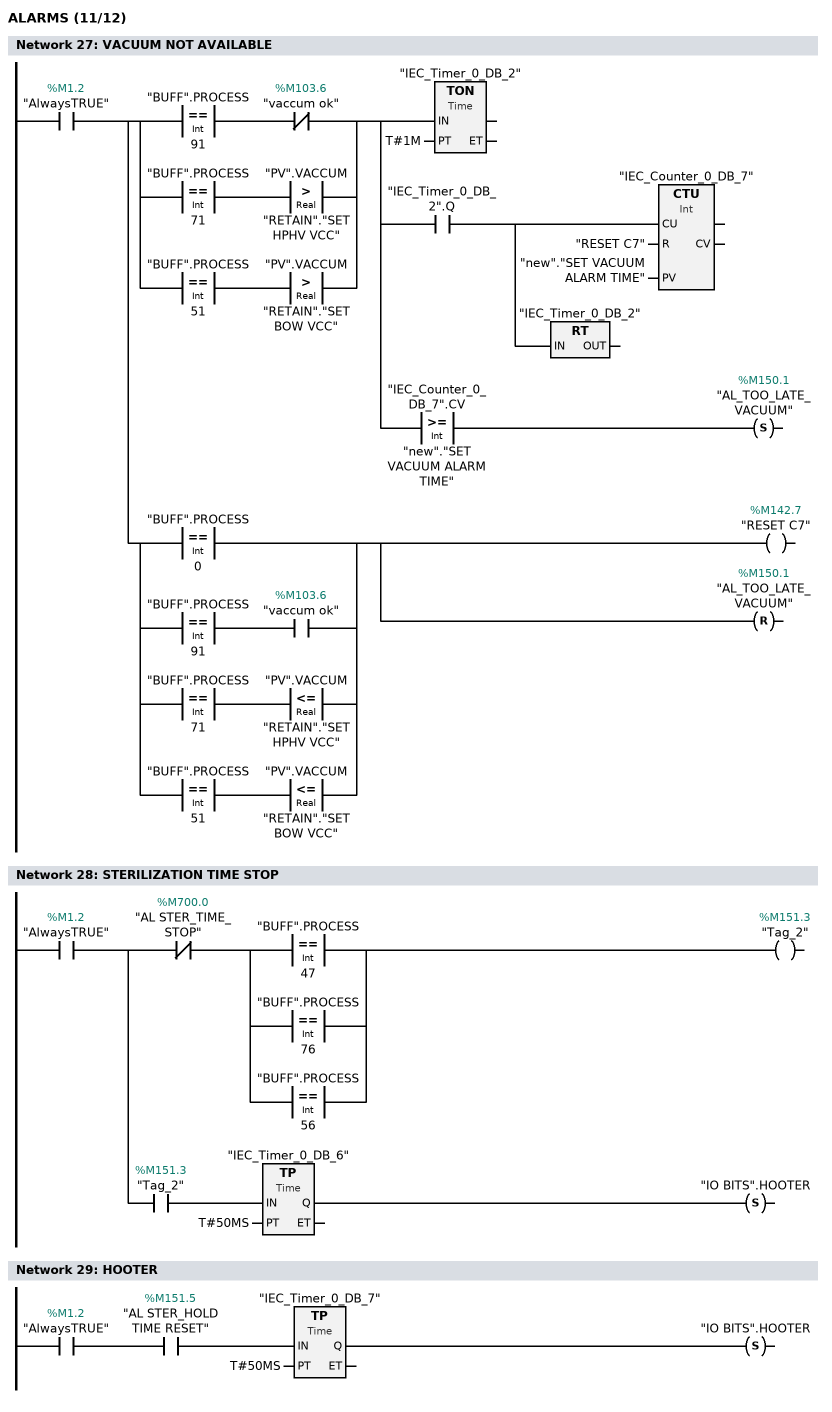
   RUNG wire#powerrail
      Contact( "AlwaysTRUE" )
      wire#w1
      { S7_Templates := "SrcType := Int" } EQ_Contact(in1 := "BUFF".PROCESS, in2 := 91)
      I_Contact( "vaccum ok" )
      wire#w2
      { S7_Templates := "time_type := Time" } "IEC_Timer_0_DB_2".TON(pt := T#1M, et =>)
   END_RUNG
   RUNG wire#w1
      { S7_Templates := "SrcType := Int" } EQ_Contact(in1 := "BUFF".PROCESS, in2 := 71)
      { S7_Templates := "SrcType := Real" } GT_Contact(in1 := "PV".VACCUM, in2 := "RETAIN"."SET HPHV VCC")
   END_RUNG wire#w2
   RUNG wire#w1
      { S7_Templates := "SrcType := Int" } EQ_Contact(in1 := "BUFF".PROCESS, in2 := 51)
      { S7_Templates := "SrcType := Real" } GT_Contact(in1 := "PV".VACCUM, in2 := "RETAIN"."SET BOW VCC")
   END_RUNG wire#w2
   RUNG wire#w2
      Contact( "IEC_Timer_0_DB_2".Q )
      wire#w3
      { S7_Templates := "value_type := Int" } "IEC_Counter_0_DB_7".CTU(r := "RESET C7", pv := "new"."SET VACUUM ALARM TIME", cv =>)
   END_RUNG
   RUNG wire#w3
      RT_Coil( "IEC_Timer_0_DB_2" )
   END_RUNG
   RUNG wire#w2
      { S7_Templates := "SrcType := Int" } GE_Contact(in1 := "IEC_Counter_0_DB_7".CV, in2 := "new"."SET VACUUM ALARM TIME")
      S_Coil( "AL_TOO_LATE_VACUUM" )
   END_RUNG
   RUNG wire#w1
      { S7_Templates := "SrcType := Int" } EQ_Contact(in1 := "BUFF".PROCESS, in2 := 0)
      wire#w4
      Coil( "RESET C7" )
   END_RUNG
   RUNG wire#w1
      { S7_Templates := "SrcType := Int" } EQ_Contact(in1 := "BUFF".PROCESS, in2 := 91)
      Contact( "vaccum ok" )
   END_RUNG wire#w4
   RUNG wire#w1
      { S7_Templates := "SrcType := Int" } EQ_Contact(in1 := "BUFF".PROCESS, in2 := 71)
      { S7_Templates := "SrcType := Real" } LE_Contact(in1 := "PV".VACCUM, in2 := "RETAIN"."SET HPHV VCC")
   END_RUNG wire#w4
   RUNG wire#w1
      { S7_Templates := "SrcType := Int" } EQ_Contact(in1 := "BUFF".PROCESS, in2 := 51)
      { S7_Templates := "SrcType := Real" } LE_Contact(in1 := "PV".VACCUM, in2 := "RETAIN"."SET BOW VCC")
   END_RUNG wire#w4
   RUNG wire#w4
      R_Coil( "AL_TOO_LATE_VACUUM" )
   END_RUNG
   // the same network as SCL:
   #_w1 := "AlwaysTRUE" AND ((("BUFF".PROCESS = 91) AND NOT "vaccum ok") OR (("BUFF".PROCESS = 71) AND ("PV".VACCUM > "RETAIN"."SET HPHV VCC")) OR (("BUFF".PROCESS = 51) AND ("PV".VACCUM > "RETAIN"."SET BOW VCC")));
   "IEC_Timer_0_DB_2".TON(IN := #_w1, PT := T#1M);
   #_w2 := #_w1 AND "IEC_Timer_0_DB_2".Q;
   "IEC_Counter_0_DB_7".CTU(CU := #_w2, R := "RESET C7", PV := "new"."SET VACUUM ALARM TIME");
   IF #_w2 THEN RESET_TIMER("IEC_Timer_0_DB_2"); END_IF;
   IF #_w1 AND ("IEC_Counter_0_DB_7".CV >= "new"."SET VACUUM ALARM TIME") THEN
       "AL_TOO_LATE_VACUUM" := TRUE;
   END_IF;
   "RESET C7" := "AlwaysTRUE" AND (("BUFF".PROCESS = 0) OR (("BUFF".PROCESS = 91) AND "vaccum ok") OR (("BUFF".PROCESS = 71) AND ("PV".VACCUM <= "RETAIN"."SET HPHV VCC")) OR (("BUFF".PROCESS = 51) AND ("PV".VACCUM <= "RETAIN"."SET BOW VCC")));
   IF "RESET C7" THEN "AL_TOO_LATE_VACUUM" := FALSE; END_IF;
END_REGION

REGION Network 28: STERILIZATION TIME STOP
   RUNG wire#powerrail
      Contact( "AlwaysTRUE" )
      wire#w1
      I_Contact( "AL STER_TIME_STOP" )
      wire#w2
      { S7_Templates := "SrcType := Int" } EQ_Contact(in1 := "BUFF".PROCESS, in2 := 47)
      wire#w3
      Coil( "Tag_2" )
   END_RUNG
   RUNG wire#w2
      { S7_Templates := "SrcType := Int" } EQ_Contact(in1 := "BUFF".PROCESS, in2 := 76)
   END_RUNG wire#w3
   RUNG wire#w2
      { S7_Templates := "SrcType := Int" } EQ_Contact(in1 := "BUFF".PROCESS, in2 := 56)
   END_RUNG wire#w3
   RUNG wire#w1
      Contact( "Tag_2" )
      { S7_Templates := "time_type := Time" } "IEC_Timer_0_DB_6".TP(pt := T#50MS, et =>)
      S_Coil( "IO BITS".HOOTER )
   END_RUNG
   // the same network as SCL:
   "Tag_2" := "AlwaysTRUE" AND NOT "AL STER_TIME_STOP" AND (("BUFF".PROCESS = 47) OR ("BUFF".PROCESS = 76) OR ("BUFF".PROCESS = 56));
   "IEC_Timer_0_DB_6".TP(IN := "AlwaysTRUE" AND "Tag_2", PT := T#50MS);
   IF "IEC_Timer_0_DB_6".Q THEN "IO BITS".HOOTER := TRUE; END_IF;
END_REGION

REGION Network 29: HOOTER
   RUNG wire#powerrail
      Contact( "AlwaysTRUE" )
      Contact( "AL STER_HOLD TIME RESET" )
      { S7_Templates := "time_type := Time" } "IEC_Timer_0_DB_7".TP(pt := T#50MS, et =>)
      S_Coil( "IO BITS".HOOTER )
   END_RUNG
   // the same network as SCL:
   "IEC_Timer_0_DB_7".TP(IN := "AlwaysTRUE" AND "AL STER_HOLD TIME RESET", PT := T#50MS);
   IF "IEC_Timer_0_DB_7".Q THEN "IO BITS".HOOTER := TRUE; END_IF;
END_REGION

REGION Network 30: boiler water level low
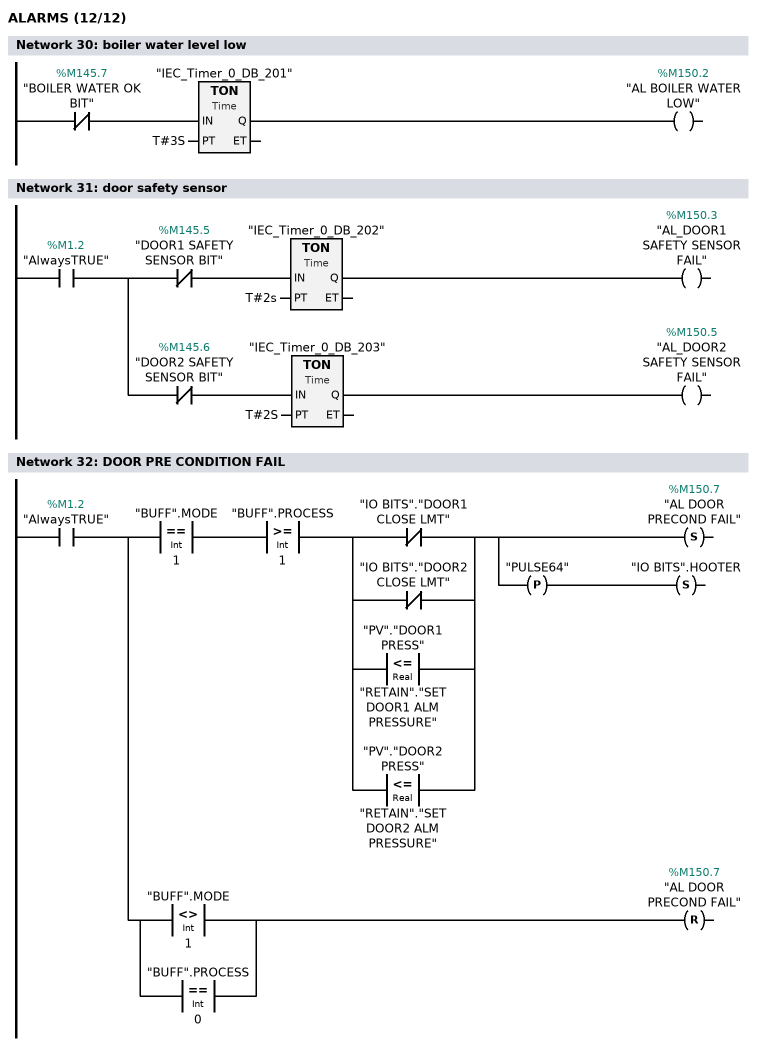
   RUNG wire#powerrail
      I_Contact( "BOILER WATER OK BIT" )
      { S7_Templates := "time_type := Time" } "IEC_Timer_0_DB_201".TON(pt := T#3S, et =>)
      Coil( "AL BOILER WATER LOW" )
   END_RUNG
   // the same network as SCL:
   "IEC_Timer_0_DB_201".TON(IN := NOT "BOILER WATER OK BIT", PT := T#3S);
   "AL BOILER WATER LOW" := "IEC_Timer_0_DB_201".Q;
END_REGION

REGION Network 31: door safety sensor
   RUNG wire#powerrail
      Contact( "AlwaysTRUE" )
      wire#w1
      I_Contact( "DOOR1 SAFETY SENSOR BIT" )
      { S7_Templates := "time_type := Time" } "IEC_Timer_0_DB_202".TON(pt := T#2s, et =>)
      Coil( "AL_DOOR1 SAFETY SENSOR FAIL" )
   END_RUNG
   RUNG wire#w1
      I_Contact( "DOOR2 SAFETY SENSOR BIT" )
      { S7_Templates := "time_type := Time" } "IEC_Timer_0_DB_203".TON(pt := T#2S, et =>)
      Coil( "AL_DOOR2 SAFETY SENSOR FAIL" )
   END_RUNG
   // the same network as SCL:
   "IEC_Timer_0_DB_202".TON(IN := "AlwaysTRUE" AND NOT "DOOR1 SAFETY SENSOR BIT", PT := T#2s);
   "AL_DOOR1 SAFETY SENSOR FAIL" := "IEC_Timer_0_DB_202".Q;
   "IEC_Timer_0_DB_203".TON(IN := "AlwaysTRUE" AND NOT "DOOR2 SAFETY SENSOR BIT", PT := T#2S);
   "AL_DOOR2 SAFETY SENSOR FAIL" := "IEC_Timer_0_DB_203".Q;
END_REGION

REGION Network 32: DOOR PRE CONDITION FAIL
   RUNG wire#powerrail
      Contact( "AlwaysTRUE" )
      wire#w1
      { S7_Templates := "SrcType := Int" } EQ_Contact(in1 := "BUFF".MODE, in2 := 1)
      { S7_Templates := "SrcType := Int" } GE_Contact(in1 := "BUFF".PROCESS, in2 := 1)
      wire#w2
      I_Contact( "IO BITS"."DOOR1 CLOSE LMT" )
      wire#w3
      S_Coil( "AL DOOR PRECOND FAIL" )
   END_RUNG
   RUNG wire#w2
      I_Contact( "IO BITS"."DOOR2 CLOSE LMT" )
   END_RUNG wire#w3
   RUNG wire#w2
      { S7_Templates := "SrcType := Real" } LE_Contact(in1 := "PV"."DOOR1 PRESS", in2 := "RETAIN"."SET DOOR1 ALM PRESSURE")
   END_RUNG wire#w3
   RUNG wire#w2
      { S7_Templates := "SrcType := Real" } LE_Contact(in1 := "PV"."DOOR2 PRESS", in2 := "RETAIN"."SET DOOR2 ALM PRESSURE")
   END_RUNG wire#w3
   RUNG wire#w3
      P_Trig( "PULSE64" )
      S_Coil( "IO BITS".HOOTER )
   END_RUNG
   RUNG wire#w1
      { S7_Templates := "SrcType := Int" } NE_Contact(in1 := "BUFF".MODE, in2 := 1)
      wire#w4
      R_Coil( "AL DOOR PRECOND FAIL" )
   END_RUNG
   RUNG wire#w1
      { S7_Templates := "SrcType := Int" } EQ_Contact(in1 := "BUFF".PROCESS, in2 := 0)
   END_RUNG wire#w4
   // the same network as SCL:
   #_w1 := "AlwaysTRUE" AND ("BUFF".MODE = 1) AND ("BUFF".PROCESS >= 1) AND (NOT "IO BITS"."DOOR1 CLOSE LMT" OR NOT "IO BITS"."DOOR2 CLOSE LMT" OR ("PV"."DOOR1 PRESS" <= "RETAIN"."SET DOOR1 ALM PRESSURE") OR ("PV"."DOOR2 PRESS" <= "RETAIN"."SET DOOR2 ALM PRESSURE"));
   IF #_w1 THEN "AL DOOR PRECOND FAIL" := TRUE; END_IF;
   #_w2 := #_w1 AND NOT "PULSE64";   // rising edge
   "PULSE64" := #_w1;
   IF #_w2 THEN "IO BITS".HOOTER := TRUE; END_IF;
   IF "AlwaysTRUE" AND (("BUFF".MODE <> 1) OR ("BUFF".PROCESS = 0)) THEN
       "AL DOOR PRECOND FAIL" := FALSE;
   END_IF;
END_REGION
END_FUNCTION

FUNCTION "OUTPUT" : Void   // FC4, LAD
{ S7_Optimized_Access := 'TRUE' }
// stored: SetENOAutomatically false
   VAR_TEMP   // added for the SCL form of the ladder/FBD networks
      _w1 : Bool;
   END_VAR
BEGIN

REGION Network 1: VCC PUMP
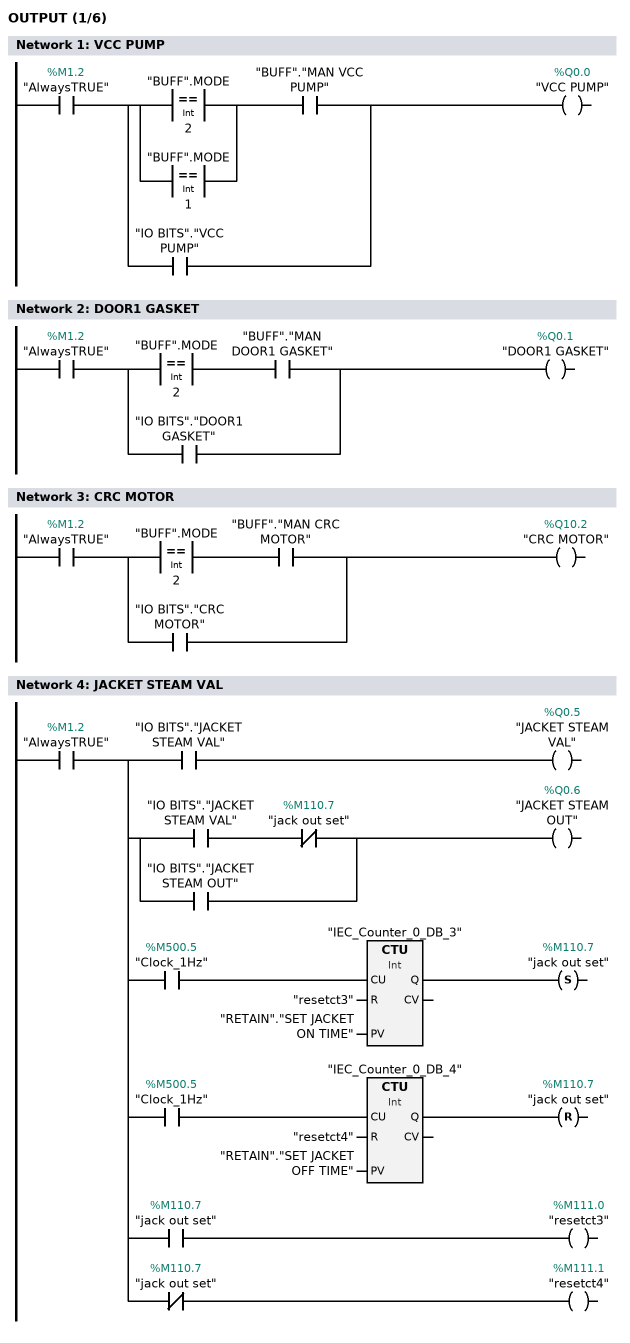
   RUNG wire#powerrail
      Contact( "AlwaysTRUE" )
      wire#w1
      { S7_Templates := "SrcType := Int" } EQ_Contact(in1 := "BUFF".MODE, in2 := 2)
      wire#w2
      Contact( "BUFF"."MAN VCC PUMP" )
      wire#w3
      Coil( "VCC PUMP" )
   END_RUNG
   RUNG wire#w1
      { S7_Templates := "SrcType := Int" } EQ_Contact(in1 := "BUFF".MODE, in2 := 1)
   END_RUNG wire#w2
   RUNG wire#w1
      Contact( "IO BITS"."VCC PUMP" )
   END_RUNG wire#w3
   // the same network as SCL:
   "VCC PUMP" := "AlwaysTRUE" AND (((("BUFF".MODE = 2) OR ("BUFF".MODE = 1)) AND "BUFF"."MAN VCC PUMP") OR "IO BITS"."VCC PUMP");
END_REGION

REGION Network 2: DOOR1 GASKET
   RUNG wire#powerrail
      Contact( "AlwaysTRUE" )
      wire#w1
      { S7_Templates := "SrcType := Int" } EQ_Contact(in1 := "BUFF".MODE, in2 := 2)
      Contact( "BUFF"."MAN DOOR1 GASKET" )
      wire#w2
      Coil( "DOOR1 GASKET" )
   END_RUNG
   RUNG wire#w1
      Contact( "IO BITS"."DOOR1 GASKET" )
   END_RUNG wire#w2
   // the same network as SCL:
   "DOOR1 GASKET" := "AlwaysTRUE" AND ((("BUFF".MODE = 2) AND "BUFF"."MAN DOOR1 GASKET") OR "IO BITS"."DOOR1 GASKET");
END_REGION

REGION Network 3: CRC MOTOR
   RUNG wire#powerrail
      Contact( "AlwaysTRUE" )
      wire#w1
      { S7_Templates := "SrcType := Int" } EQ_Contact(in1 := "BUFF".MODE, in2 := 2)
      Contact( "BUFF"."MAN CRC MOTOR" )
      wire#w2
      Coil( "CRC MOTOR" )
   END_RUNG
   RUNG wire#w1
      Contact( "IO BITS"."CRC MOTOR" )
   END_RUNG wire#w2
   // the same network as SCL:
   "CRC MOTOR" := "AlwaysTRUE" AND ((("BUFF".MODE = 2) AND "BUFF"."MAN CRC MOTOR") OR "IO BITS"."CRC MOTOR");
END_REGION

REGION Network 4: JACKET STEAM VAL
   RUNG wire#powerrail
      Contact( "AlwaysTRUE" )
      wire#w1
      Contact( "IO BITS"."JACKET STEAM VAL" )
      Coil( "JACKET STEAM VAL" )
   END_RUNG
   RUNG wire#w1
      Contact( "IO BITS"."JACKET STEAM VAL" )
      I_Contact( "jack out set" )
      wire#w2
      Coil( "JACKET STEAM OUT" )
   END_RUNG
   RUNG wire#w1
      Contact( "IO BITS"."JACKET STEAM OUT" )
   END_RUNG wire#w2
   RUNG wire#w1
      Contact( "Clock_1Hz" )
      { S7_Templates := "value_type := Int" } "IEC_Counter_0_DB_3".CTU(r := "resetct3", pv := "RETAIN"."SET JACKET ON TIME", cv =>)
      S_Coil( "jack out set" )
   END_RUNG
   RUNG wire#w1
      Contact( "Clock_1Hz" )
      { S7_Templates := "value_type := Int" } "IEC_Counter_0_DB_4".CTU(r := "resetct4", pv := "RETAIN"."SET JACKET OFF TIME", cv =>)
      R_Coil( "jack out set" )
   END_RUNG
   RUNG wire#w1
      Contact( "jack out set" )
      Coil( "resetct3" )
   END_RUNG
   RUNG wire#w1
      I_Contact( "jack out set" )
      Coil( "resetct4" )
   END_RUNG
   // the same network as SCL:
   "JACKET STEAM VAL" := "AlwaysTRUE" AND "IO BITS"."JACKET STEAM VAL";
   "JACKET STEAM OUT" := "AlwaysTRUE" AND (("IO BITS"."JACKET STEAM VAL" AND NOT "jack out set") OR "IO BITS"."JACKET STEAM OUT");
   "IEC_Counter_0_DB_3".CTU(CU := "AlwaysTRUE" AND "Clock_1Hz",
                           R := "resetct3",
                           PV := "RETAIN"."SET JACKET ON TIME");
   IF "IEC_Counter_0_DB_3".Q THEN "jack out set" := TRUE; END_IF;
   "IEC_Counter_0_DB_4".CTU(CU := "AlwaysTRUE" AND "Clock_1Hz",
                           R := "resetct4",
                           PV := "RETAIN"."SET JACKET OFF TIME");
   IF "IEC_Counter_0_DB_4".Q THEN "jack out set" := FALSE; END_IF;
   "resetct3" := "AlwaysTRUE" AND "jack out set";
   "resetct4" := "AlwaysTRUE" AND NOT "jack out set";
END_REGION

REGION Network 5: CHAMBER STEAM VAL
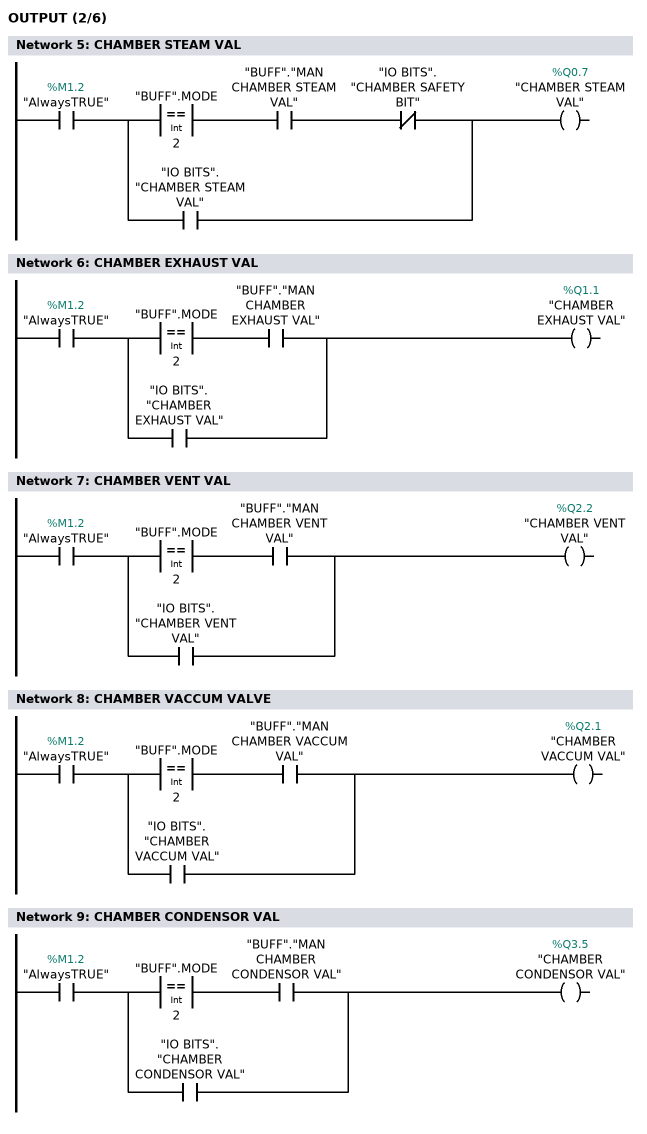
   RUNG wire#powerrail
      Contact( "AlwaysTRUE" )
      wire#w1
      { S7_Templates := "SrcType := Int" } EQ_Contact(in1 := "BUFF".MODE, in2 := 2)
      Contact( "BUFF"."MAN CHAMBER STEAM VAL" )
      I_Contact( "IO BITS"."CHAMBER SAFETY BIT" )
      wire#w2
      Coil( "CHAMBER STEAM VAL" )
   END_RUNG
   RUNG wire#w1
      Contact( "IO BITS"."CHAMBER STEAM VAL" )
   END_RUNG wire#w2
   // the same network as SCL:
   "CHAMBER STEAM VAL" := "AlwaysTRUE" AND ((("BUFF".MODE = 2) AND "BUFF"."MAN CHAMBER STEAM VAL" AND NOT "IO BITS"."CHAMBER SAFETY BIT") OR "IO BITS"."CHAMBER STEAM VAL");
END_REGION

REGION Network 6: CHAMBER EXHAUST VAL
   RUNG wire#powerrail
      Contact( "AlwaysTRUE" )
      wire#w1
      { S7_Templates := "SrcType := Int" } EQ_Contact(in1 := "BUFF".MODE, in2 := 2)
      Contact( "BUFF"."MAN CHAMBER EXHAUST VAL" )
      wire#w2
      Coil( "CHAMBER EXHAUST VAL" )
   END_RUNG
   RUNG wire#w1
      Contact( "IO BITS"."CHAMBER EXHAUST VAL" )
   END_RUNG wire#w2
   // the same network as SCL:
   "CHAMBER EXHAUST VAL" := "AlwaysTRUE" AND ((("BUFF".MODE = 2) AND "BUFF"."MAN CHAMBER EXHAUST VAL") OR "IO BITS"."CHAMBER EXHAUST VAL");
END_REGION

REGION Network 7: CHAMBER VENT VAL
   RUNG wire#powerrail
      Contact( "AlwaysTRUE" )
      wire#w1
      { S7_Templates := "SrcType := Int" } EQ_Contact(in1 := "BUFF".MODE, in2 := 2)
      Contact( "BUFF"."MAN CHAMBER VENT VAL" )
      wire#w2
      Coil( "CHAMBER VENT VAL" )
   END_RUNG
   RUNG wire#w1
      Contact( "IO BITS"."CHAMBER VENT VAL" )
   END_RUNG wire#w2
   // the same network as SCL:
   "CHAMBER VENT VAL" := "AlwaysTRUE" AND ((("BUFF".MODE = 2) AND "BUFF"."MAN CHAMBER VENT VAL") OR "IO BITS"."CHAMBER VENT VAL");
END_REGION

REGION Network 8: CHAMBER VACCUM VALVE
   RUNG wire#powerrail
      Contact( "AlwaysTRUE" )
      wire#w1
      { S7_Templates := "SrcType := Int" } EQ_Contact(in1 := "BUFF".MODE, in2 := 2)
      Contact( "BUFF"."MAN CHAMBER VACCUM VAL" )
      wire#w2
      Coil( "CHAMBER VACCUM VAL" )
   END_RUNG
   RUNG wire#w1
      Contact( "IO BITS"."CHAMBER VACCUM VAL" )
   END_RUNG wire#w2
   // the same network as SCL:
   "CHAMBER VACCUM VAL" := "AlwaysTRUE" AND ((("BUFF".MODE = 2) AND "BUFF"."MAN CHAMBER VACCUM VAL") OR "IO BITS"."CHAMBER VACCUM VAL");
END_REGION

REGION Network 9: CHAMBER CONDENSOR VAL
   RUNG wire#powerrail
      Contact( "AlwaysTRUE" )
      wire#w1
      { S7_Templates := "SrcType := Int" } EQ_Contact(in1 := "BUFF".MODE, in2 := 2)
      Contact( "BUFF"."MAN CHAMBER CONDENSOR VAL" )
      wire#w2
      Coil( "CHAMBER CONDENSOR VAL" )
   END_RUNG
   RUNG wire#w1
      Contact( "IO BITS"."CHAMBER CONDENSOR VAL" )
   END_RUNG wire#w2
   // the same network as SCL:
   "CHAMBER CONDENSOR VAL" := "AlwaysTRUE" AND ((("BUFF".MODE = 2) AND "BUFF"."MAN CHAMBER CONDENSOR VAL") OR "IO BITS"."CHAMBER CONDENSOR VAL");
END_REGION

REGION Network 10: process on lamp
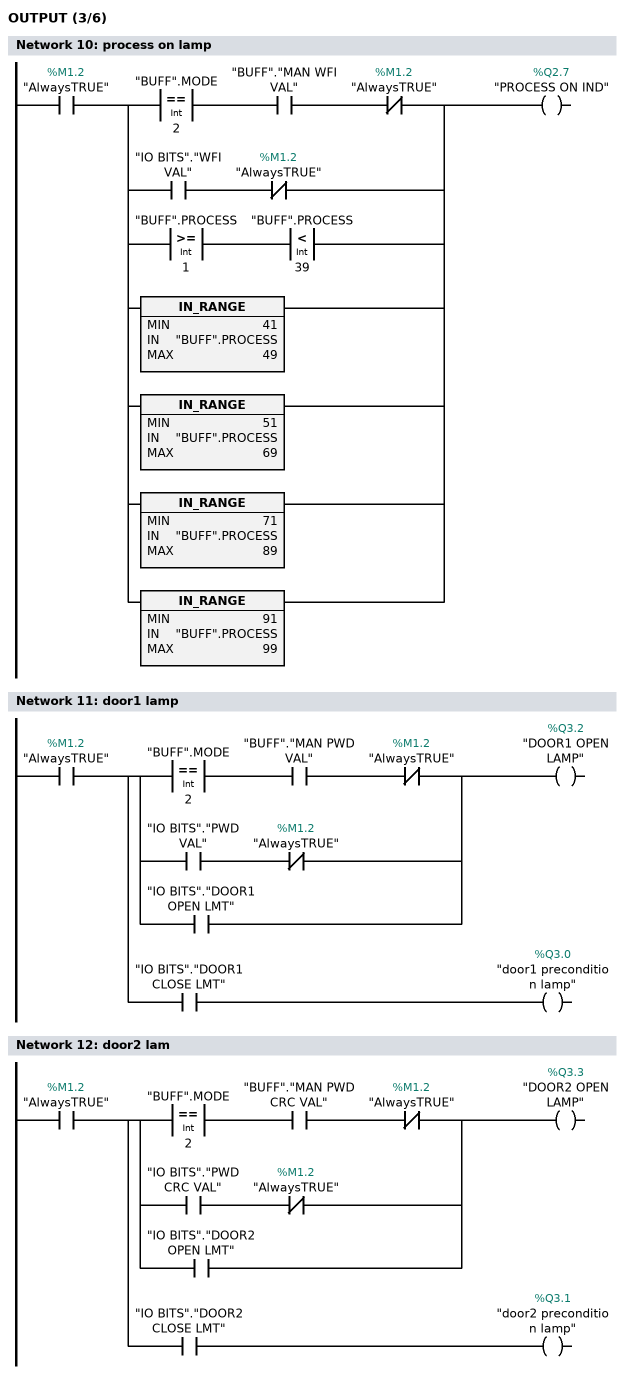
   RUNG wire#powerrail
      Contact( "AlwaysTRUE" )
      wire#w1
      { S7_Templates := "SrcType := Int" } EQ_Contact(in1 := "BUFF".MODE, in2 := 2)
      Contact( "BUFF"."MAN WFI VAL" )
      I_Contact( "AlwaysTRUE" )
      wire#w2
      Coil( "PROCESS ON IND" )
   END_RUNG
   RUNG wire#w1
      Contact( "IO BITS"."WFI VAL" )
      I_Contact( "AlwaysTRUE" )
   END_RUNG wire#w2
   RUNG wire#w1
      { S7_Templates := "SrcType := Int" } GE_Contact(in1 := "BUFF".PROCESS, in2 := 1)
      { S7_Templates := "SrcType := Int" } LT_Contact(in1 := "BUFF".PROCESS, in2 := 39)
   END_RUNG wire#w2
   RUNG wire#w1
      { S7_Templates := "SrcType := Int" } InRange(min := 41, in := "BUFF".PROCESS, max := 49)
   END_RUNG wire#w2
   RUNG wire#w1
      { S7_Templates := "SrcType := Int" } InRange(min := 51, in := "BUFF".PROCESS, max := 69)
   END_RUNG wire#w2
   RUNG wire#w1
      { S7_Templates := "SrcType := Int" } InRange(min := 71, in := "BUFF".PROCESS, max := 89)
   END_RUNG wire#w2
   RUNG wire#w1
      { S7_Templates := "SrcType := Int" } InRange(min := 91, in := "BUFF".PROCESS, max := 99)
   END_RUNG wire#w2
   // the same network as SCL:
   "PROCESS ON IND" := "AlwaysTRUE" AND ((("BUFF".MODE = 2) AND "BUFF"."MAN WFI VAL" AND NOT "AlwaysTRUE") OR ("IO BITS"."WFI VAL" AND NOT "AlwaysTRUE") OR (("BUFF".PROCESS >= 1) AND ("BUFF".PROCESS < 39)) OR ((41 <= "BUFF".PROCESS) AND ("BUFF".PROCESS <= 49)) OR ((51 <= "BUFF".PROCESS) AND ("BUFF".PROCESS <= 69)) OR ((71 <= "BUFF".PROCESS) AND ("BUFF".PROCESS <= 89)) OR ((91 <= "BUFF".PROCESS) AND ("BUFF".PROCESS <= 99)));
END_REGION

REGION Network 11: door1 lamp
   RUNG wire#powerrail
      Contact( "AlwaysTRUE" )
      wire#w1
      { S7_Templates := "SrcType := Int" } EQ_Contact(in1 := "BUFF".MODE, in2 := 2)
      Contact( "BUFF"."MAN PWD VAL" )
      I_Contact( "AlwaysTRUE" )
      wire#w2
      Coil( "DOOR1 OPEN LAMP" )
   END_RUNG
   RUNG wire#w1
      Contact( "IO BITS"."PWD VAL" )
      I_Contact( "AlwaysTRUE" )
   END_RUNG wire#w2
   RUNG wire#w1
      Contact( "IO BITS"."DOOR1 OPEN LMT" )
   END_RUNG wire#w2
   RUNG wire#w1
      Contact( "IO BITS"."DOOR1 CLOSE LMT" )
      Coil( "door1 precondition lamp" )
   END_RUNG
   // the same network as SCL:
   "DOOR1 OPEN LAMP" := "AlwaysTRUE" AND ((("BUFF".MODE = 2) AND "BUFF"."MAN PWD VAL" AND NOT "AlwaysTRUE") OR ("IO BITS"."PWD VAL" AND NOT "AlwaysTRUE") OR "IO BITS"."DOOR1 OPEN LMT");
   "door1 precondition lamp" := "AlwaysTRUE" AND "IO BITS"."DOOR1 CLOSE LMT";
END_REGION

REGION Network 12: door2 lam
   RUNG wire#powerrail
      Contact( "AlwaysTRUE" )
      wire#w1
      { S7_Templates := "SrcType := Int" } EQ_Contact(in1 := "BUFF".MODE, in2 := 2)
      Contact( "BUFF"."MAN PWD CRC VAL" )
      I_Contact( "AlwaysTRUE" )
      wire#w2
      Coil( "DOOR2 OPEN LAMP" )
   END_RUNG
   RUNG wire#w1
      Contact( "IO BITS"."PWD CRC VAL" )
      I_Contact( "AlwaysTRUE" )
   END_RUNG wire#w2
   RUNG wire#w1
      Contact( "IO BITS"."DOOR2 OPEN LMT" )
   END_RUNG wire#w2
   RUNG wire#w1
      Contact( "IO BITS"."DOOR2 CLOSE LMT" )
      Coil( "door2 precondition lamp" )
   END_RUNG
   // the same network as SCL:
   "DOOR2 OPEN LAMP" := "AlwaysTRUE" AND ((("BUFF".MODE = 2) AND "BUFF"."MAN PWD CRC VAL" AND NOT "AlwaysTRUE") OR ("IO BITS"."PWD CRC VAL" AND NOT "AlwaysTRUE") OR "IO BITS"."DOOR2 OPEN LMT");
   "door2 precondition lamp" := "AlwaysTRUE" AND "IO BITS"."DOOR2 CLOSE LMT";
END_REGION

REGION Network 13: DETERGENT DSG VAL
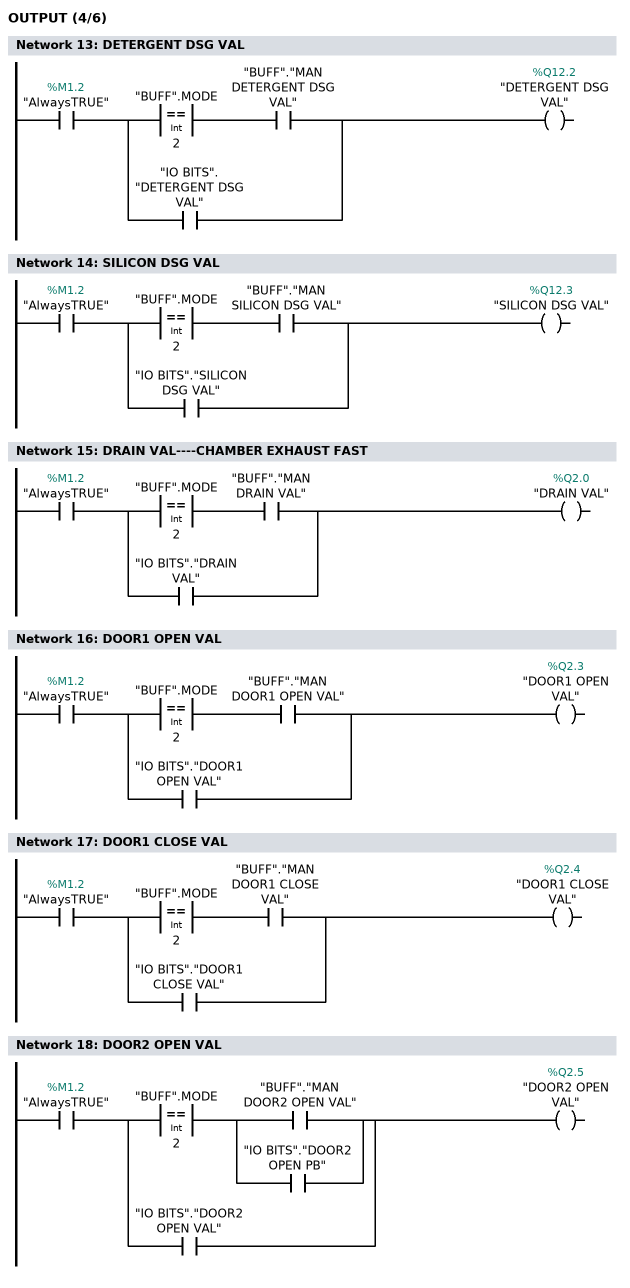
   RUNG wire#powerrail
      Contact( "AlwaysTRUE" )
      wire#w1
      { S7_Templates := "SrcType := Int" } EQ_Contact(in1 := "BUFF".MODE, in2 := 2)
      Contact( "BUFF"."MAN DETERGENT DSG VAL" )
      wire#w2
      Coil( "DETERGENT DSG VAL" )
   END_RUNG
   RUNG wire#w1
      Contact( "IO BITS"."DETERGENT DSG VAL" )
   END_RUNG wire#w2
   // the same network as SCL:
   "DETERGENT DSG VAL" := "AlwaysTRUE" AND ((("BUFF".MODE = 2) AND "BUFF"."MAN DETERGENT DSG VAL") OR "IO BITS"."DETERGENT DSG VAL");
END_REGION

REGION Network 14: SILICON DSG VAL
   RUNG wire#powerrail
      Contact( "AlwaysTRUE" )
      wire#w1
      { S7_Templates := "SrcType := Int" } EQ_Contact(in1 := "BUFF".MODE, in2 := 2)
      Contact( "BUFF"."MAN SILICON DSG VAL" )
      wire#w2
      Coil( "SILICON DSG VAL" )
   END_RUNG
   RUNG wire#w1
      Contact( "IO BITS"."SILICON DSG VAL" )
   END_RUNG wire#w2
   // the same network as SCL:
   "SILICON DSG VAL" := "AlwaysTRUE" AND ((("BUFF".MODE = 2) AND "BUFF"."MAN SILICON DSG VAL") OR "IO BITS"."SILICON DSG VAL");
END_REGION

REGION Network 15: DRAIN VAL----CHAMBER EXHAUST FAST
   RUNG wire#powerrail
      Contact( "AlwaysTRUE" )
      wire#w1
      { S7_Templates := "SrcType := Int" } EQ_Contact(in1 := "BUFF".MODE, in2 := 2)
      Contact( "BUFF"."MAN DRAIN VAL" )
      wire#w2
      Coil( "DRAIN VAL" )
   END_RUNG
   RUNG wire#w1
      Contact( "IO BITS"."DRAIN VAL" )
   END_RUNG wire#w2
   // the same network as SCL:
   "DRAIN VAL" := "AlwaysTRUE" AND ((("BUFF".MODE = 2) AND "BUFF"."MAN DRAIN VAL") OR "IO BITS"."DRAIN VAL");
END_REGION

REGION Network 16: DOOR1 OPEN VAL
   RUNG wire#powerrail
      Contact( "AlwaysTRUE" )
      wire#w1
      { S7_Templates := "SrcType := Int" } EQ_Contact(in1 := "BUFF".MODE, in2 := 2)
      Contact( "BUFF"."MAN DOOR1 OPEN VAL" )
      wire#w2
      Coil( "DOOR1 OPEN VAL" )
   END_RUNG
   RUNG wire#w1
      Contact( "IO BITS"."DOOR1 OPEN VAL" )
   END_RUNG wire#w2
   // the same network as SCL:
   "DOOR1 OPEN VAL" := "AlwaysTRUE" AND ((("BUFF".MODE = 2) AND "BUFF"."MAN DOOR1 OPEN VAL") OR "IO BITS"."DOOR1 OPEN VAL");
END_REGION

REGION Network 17: DOOR1 CLOSE VAL
   RUNG wire#powerrail
      Contact( "AlwaysTRUE" )
      wire#w1
      { S7_Templates := "SrcType := Int" } EQ_Contact(in1 := "BUFF".MODE, in2 := 2)
      Contact( "BUFF"."MAN DOOR1 CLOSE VAL" )
      wire#w2
      Coil( "DOOR1 CLOSE VAL" )
   END_RUNG
   RUNG wire#w1
      Contact( "IO BITS"."DOOR1 CLOSE VAL" )
   END_RUNG wire#w2
   // the same network as SCL:
   "DOOR1 CLOSE VAL" := "AlwaysTRUE" AND ((("BUFF".MODE = 2) AND "BUFF"."MAN DOOR1 CLOSE VAL") OR "IO BITS"."DOOR1 CLOSE VAL");
END_REGION

REGION Network 18: DOOR2 OPEN VAL
   RUNG wire#powerrail
      Contact( "AlwaysTRUE" )
      wire#w1
      { S7_Templates := "SrcType := Int" } EQ_Contact(in1 := "BUFF".MODE, in2 := 2)
      wire#w2
      Contact( "BUFF"."MAN DOOR2 OPEN VAL" )
      wire#w3
      Coil( "DOOR2 OPEN VAL" )
   END_RUNG
   RUNG wire#w2
      Contact( "IO BITS"."DOOR2 OPEN PB" )
   END_RUNG wire#w3
   RUNG wire#w1
      Contact( "IO BITS"."DOOR2 OPEN VAL" )
   END_RUNG wire#w3
   // the same network as SCL:
   "DOOR2 OPEN VAL" := "AlwaysTRUE" AND ((("BUFF".MODE = 2) AND ("BUFF"."MAN DOOR2 OPEN VAL" OR "IO BITS"."DOOR2 OPEN PB")) OR "IO BITS"."DOOR2 OPEN VAL");
END_REGION

REGION Network 19: DOOR2 CLOSE VAL
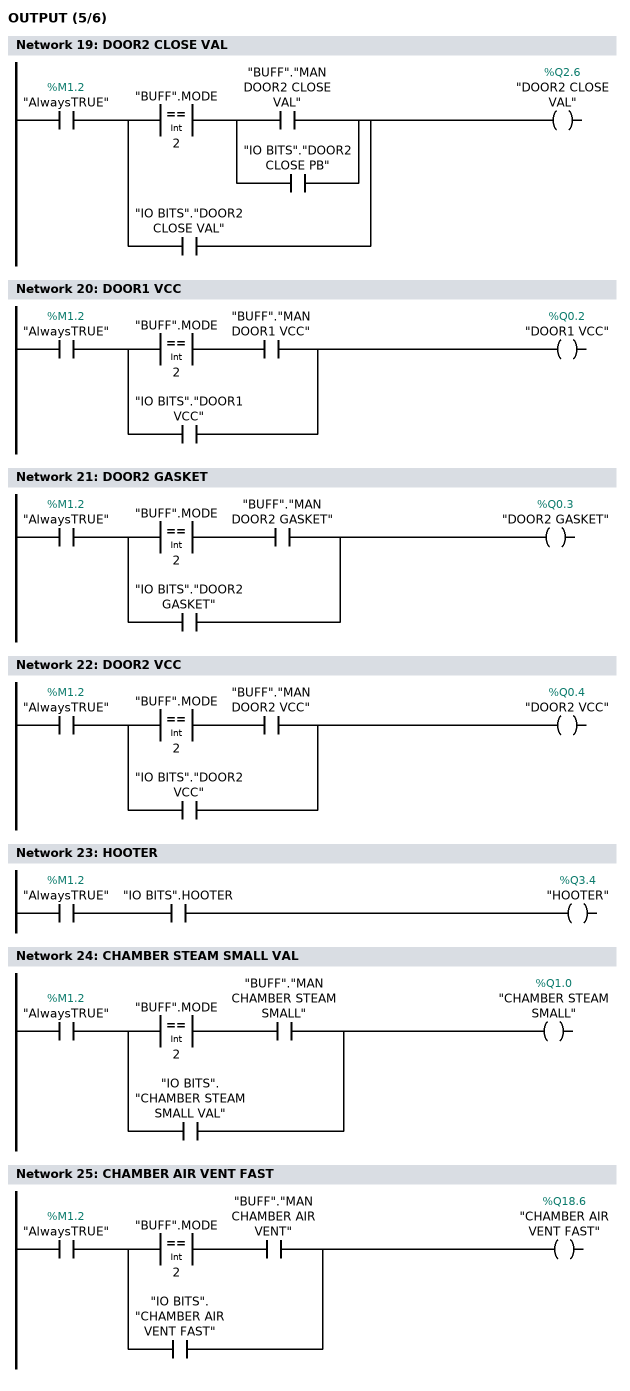
   RUNG wire#powerrail
      Contact( "AlwaysTRUE" )
      wire#w1
      { S7_Templates := "SrcType := Int" } EQ_Contact(in1 := "BUFF".MODE, in2 := 2)
      wire#w2
      Contact( "BUFF"."MAN DOOR2 CLOSE VAL" )
      wire#w3
      Coil( "DOOR2 CLOSE VAL" )
   END_RUNG
   RUNG wire#w2
      Contact( "IO BITS"."DOOR2 CLOSE PB" )
   END_RUNG wire#w3
   RUNG wire#w1
      Contact( "IO BITS"."DOOR2 CLOSE VAL" )
   END_RUNG wire#w3
   // the same network as SCL:
   "DOOR2 CLOSE VAL" := "AlwaysTRUE" AND ((("BUFF".MODE = 2) AND ("BUFF"."MAN DOOR2 CLOSE VAL" OR "IO BITS"."DOOR2 CLOSE PB")) OR "IO BITS"."DOOR2 CLOSE VAL");
END_REGION

REGION Network 20: DOOR1 VCC
   RUNG wire#powerrail
      Contact( "AlwaysTRUE" )
      wire#w1
      { S7_Templates := "SrcType := Int" } EQ_Contact(in1 := "BUFF".MODE, in2 := 2)
      Contact( "BUFF"."MAN DOOR1 VCC" )
      wire#w2
      Coil( "DOOR1 VCC" )
   END_RUNG
   RUNG wire#w1
      Contact( "IO BITS"."DOOR1 VCC" )
   END_RUNG wire#w2
   // the same network as SCL:
   "DOOR1 VCC" := "AlwaysTRUE" AND ((("BUFF".MODE = 2) AND "BUFF"."MAN DOOR1 VCC") OR "IO BITS"."DOOR1 VCC");
END_REGION

REGION Network 21: DOOR2 GASKET
   RUNG wire#powerrail
      Contact( "AlwaysTRUE" )
      wire#w1
      { S7_Templates := "SrcType := Int" } EQ_Contact(in1 := "BUFF".MODE, in2 := 2)
      Contact( "BUFF"."MAN DOOR2 GASKET" )
      wire#w2
      Coil( "DOOR2 GASKET" )
   END_RUNG
   RUNG wire#w1
      Contact( "IO BITS"."DOOR2 GASKET" )
   END_RUNG wire#w2
   // the same network as SCL:
   "DOOR2 GASKET" := "AlwaysTRUE" AND ((("BUFF".MODE = 2) AND "BUFF"."MAN DOOR2 GASKET") OR "IO BITS"."DOOR2 GASKET");
END_REGION

REGION Network 22: DOOR2 VCC
   RUNG wire#powerrail
      Contact( "AlwaysTRUE" )
      wire#w1
      { S7_Templates := "SrcType := Int" } EQ_Contact(in1 := "BUFF".MODE, in2 := 2)
      Contact( "BUFF"."MAN DOOR2 VCC" )
      wire#w2
      Coil( "DOOR2 VCC" )
   END_RUNG
   RUNG wire#w1
      Contact( "IO BITS"."DOOR2 VCC" )
   END_RUNG wire#w2
   // the same network as SCL:
   "DOOR2 VCC" := "AlwaysTRUE" AND ((("BUFF".MODE = 2) AND "BUFF"."MAN DOOR2 VCC") OR "IO BITS"."DOOR2 VCC");
END_REGION

REGION Network 23: HOOTER
   RUNG wire#powerrail
      Contact( "AlwaysTRUE" )
      Contact( "IO BITS".HOOTER )
      Coil( "HOOTER" )
   END_RUNG
   // the same network as SCL:
   "HOOTER" := "AlwaysTRUE" AND "IO BITS".HOOTER;
END_REGION

REGION Network 24: CHAMBER STEAM SMALL VAL
   RUNG wire#powerrail
      Contact( "AlwaysTRUE" )
      wire#w1
      { S7_Templates := "SrcType := Int" } EQ_Contact(in1 := "BUFF".MODE, in2 := 2)
      Contact( "BUFF"."MAN CHAMBER STEAM SMALL" )
      wire#w2
      Coil( "CHAMBER STEAM SMALL" )
   END_RUNG
   RUNG wire#w1
      Contact( "IO BITS"."CHAMBER STEAM SMALL VAL" )
   END_RUNG wire#w2
   // the same network as SCL:
   "CHAMBER STEAM SMALL" := "AlwaysTRUE" AND ((("BUFF".MODE = 2) AND "BUFF"."MAN CHAMBER STEAM SMALL") OR "IO BITS"."CHAMBER STEAM SMALL VAL");
END_REGION

REGION Network 25: CHAMBER AIR VENT FAST
   RUNG wire#powerrail
      Contact( "AlwaysTRUE" )
      wire#w1
      { S7_Templates := "SrcType := Int" } EQ_Contact(in1 := "BUFF".MODE, in2 := 2)
      Contact( "BUFF"."MAN CHAMBER AIR VENT" )
      wire#w2
      Coil( "CHAMBER AIR VENT FAST" )
   END_RUNG
   RUNG wire#w1
      Contact( "IO BITS"."CHAMBER AIR VENT FAST" )
   END_RUNG wire#w2
   // the same network as SCL:
   "CHAMBER AIR VENT FAST" := "AlwaysTRUE" AND ((("BUFF".MODE = 2) AND "BUFF"."MAN CHAMBER AIR VENT") OR "IO BITS"."CHAMBER AIR VENT FAST");
END_REGION

REGION Network 26: BOILER
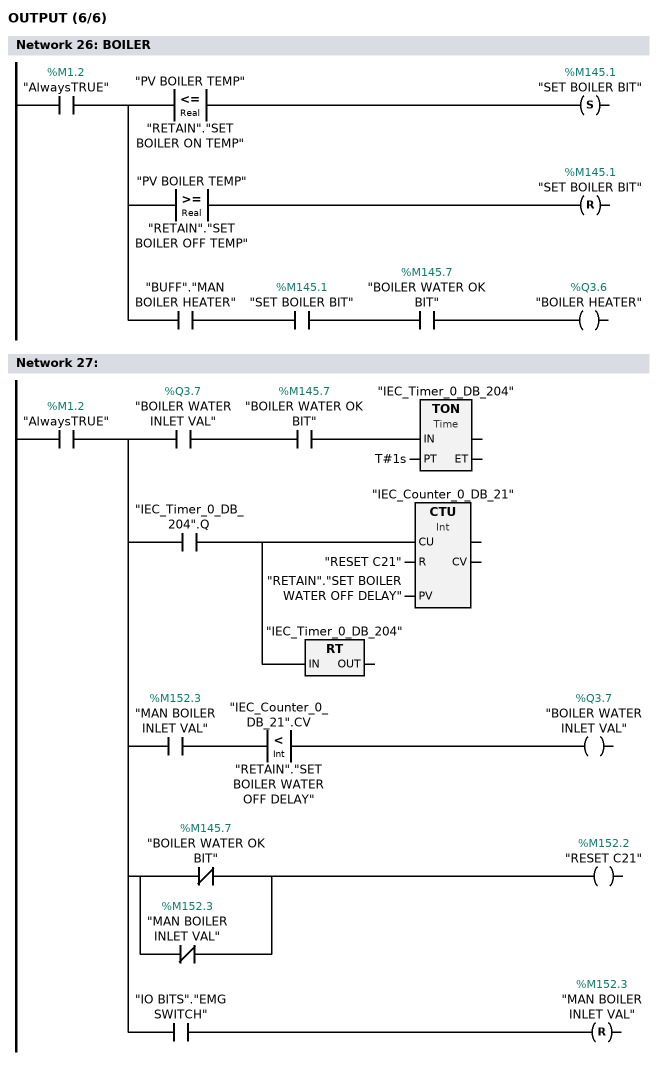
   RUNG wire#powerrail
      Contact( "AlwaysTRUE" )
      wire#w1
      { S7_Templates := "SrcType := Real" } LE_Contact(in1 := "PV BOILER TEMP", in2 := "RETAIN"."SET BOILER ON TEMP")
      S_Coil( "SET BOILER BIT" )
   END_RUNG
   RUNG wire#w1
      { S7_Templates := "SrcType := Real" } GE_Contact(in1 := "PV BOILER TEMP", in2 := "RETAIN"."SET BOILER OFF TEMP")
      R_Coil( "SET BOILER BIT" )
   END_RUNG
   RUNG wire#w1
      Contact( "BUFF"."MAN BOILER HEATER" )
      Contact( "SET BOILER BIT" )
      Contact( "BOILER WATER OK BIT" )
      Coil( "BOILER HEATER" )
   END_RUNG
   // the same network as SCL:
   IF "AlwaysTRUE" AND ("PV BOILER TEMP" <= "RETAIN"."SET BOILER ON TEMP") THEN
       "SET BOILER BIT" := TRUE;
   END_IF;
   IF "AlwaysTRUE" AND ("PV BOILER TEMP" >= "RETAIN"."SET BOILER OFF TEMP") THEN
       "SET BOILER BIT" := FALSE;
   END_IF;
   "BOILER HEATER" := "AlwaysTRUE" AND "BUFF"."MAN BOILER HEATER" AND "SET BOILER BIT" AND "BOILER WATER OK BIT";
END_REGION

REGION Network 27
   RUNG wire#powerrail
      Contact( "AlwaysTRUE" )
      wire#w1
      Contact( "BOILER WATER INLET VAL" )
      Contact( "BOILER WATER OK BIT" )
      { S7_Templates := "time_type := Time" } "IEC_Timer_0_DB_204".TON(pt := T#1s, et =>)
   END_RUNG
   RUNG wire#w1
      Contact( "IEC_Timer_0_DB_204".Q )
      wire#w2
      { S7_Templates := "value_type := Int" } "IEC_Counter_0_DB_21".CTU(r := "RESET C21", pv := "RETAIN"."SET BOILER WATER OFF DELAY", cv =>)
   END_RUNG
   RUNG wire#w2
      RT_Coil( "IEC_Timer_0_DB_204" )
   END_RUNG
   RUNG wire#w1
      Contact( "MAN BOILER INLET VAL" )
      { S7_Templates := "SrcType := Int" } LT_Contact(in1 := "IEC_Counter_0_DB_21".CV, in2 := "RETAIN"."SET BOILER WATER OFF DELAY")
      Coil( "BOILER WATER INLET VAL" )
   END_RUNG
   RUNG wire#w1
      I_Contact( "BOILER WATER OK BIT" )
      wire#w3
      Coil( "RESET C21" )
   END_RUNG
   RUNG wire#w1
      I_Contact( "MAN BOILER INLET VAL" )
   END_RUNG wire#w3
   RUNG wire#w1
      Contact( "IO BITS"."EMG SWITCH" )
      R_Coil( "MAN BOILER INLET VAL" )
   END_RUNG
   // the same network as SCL:
   "IEC_Timer_0_DB_204".TON(IN := "AlwaysTRUE" AND "BOILER WATER INLET VAL" AND "BOILER WATER OK BIT",
                           PT := T#1s);
   #_w1 := "AlwaysTRUE" AND "IEC_Timer_0_DB_204".Q;
   "IEC_Counter_0_DB_21".CTU(CU := #_w1, R := "RESET C21", PV := "RETAIN"."SET BOILER WATER OFF DELAY");
   IF #_w1 THEN RESET_TIMER("IEC_Timer_0_DB_204"); END_IF;
   "BOILER WATER INLET VAL" := "AlwaysTRUE" AND "MAN BOILER INLET VAL" AND ("IEC_Counter_0_DB_21".CV < "RETAIN"."SET BOILER WATER OFF DELAY");
   "RESET C21" := "AlwaysTRUE" AND (NOT "BOILER WATER OK BIT" OR NOT "MAN BOILER INLET VAL");
   IF "AlwaysTRUE" AND "IO BITS"."EMG SWITCH" THEN "MAN BOILER INLET VAL" := FALSE; END_IF;
END_REGION
END_FUNCTION

FUNCTION "DIG IP" : Void   // FC3, LAD
{ S7_Optimized_Access := 'TRUE' }
// stored: SetENOAutomatically false
   VAR_TEMP   // added for the SCL form of the ladder/FBD networks
      _w1 : Bool;
      _w2 : Bool;
      _w3 : Bool;
      _w4 : Bool;
      _w5 : Bool;
   END_VAR
BEGIN

REGION Network 1: BLOCK CALL
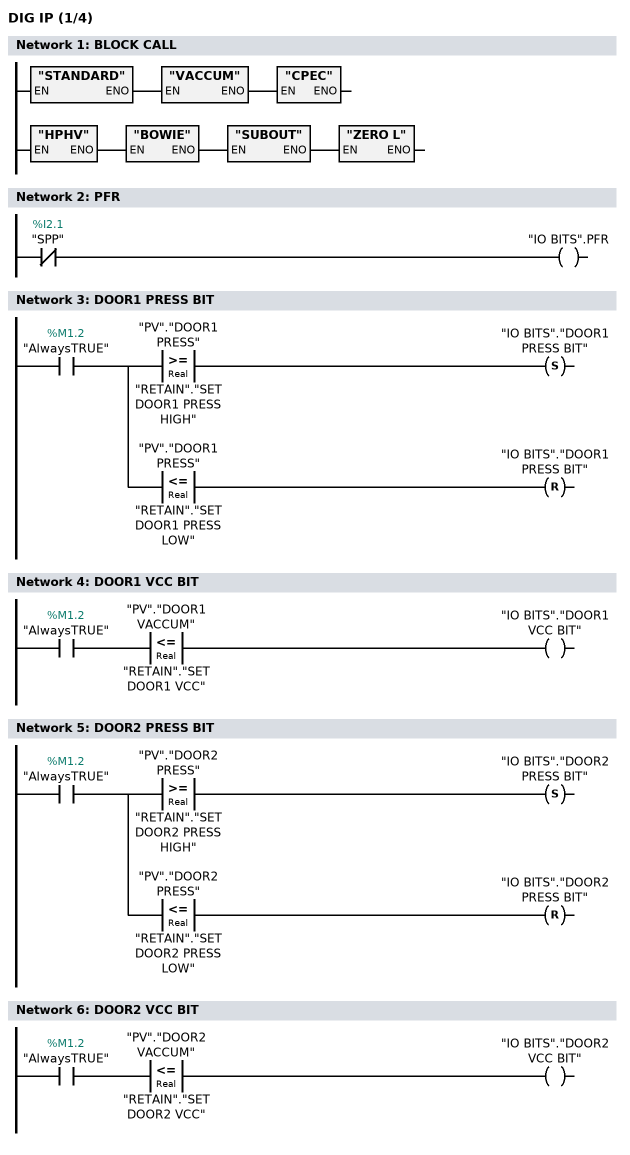
   RUNG wire#powerrail
      "STANDARD"()
      "VACCUM"()
      "CPEC"()
   END_RUNG
   RUNG wire#powerrail
      "HPHV"()
      "BOWIE"()
      "SUBOUT"()
      "ZERO L"()
   END_RUNG
   // the same network as SCL:
   "STANDARD"(ENO => #_w1);
   "VACCUM"(EN := #_w1, ENO => #_w2);
   IF #_w2 THEN "CPEC"(); END_IF;
   "HPHV"(ENO => #_w3);
   "BOWIE"(EN := #_w3, ENO => #_w4);
   "SUBOUT"(EN := #_w4, ENO => #_w5);
   IF #_w5 THEN "ZERO L"(); END_IF;
END_REGION

REGION Network 2: PFR
   RUNG wire#powerrail
      I_Contact( "SPP" )
      Coil( "IO BITS".PFR )
   END_RUNG
   // the same network as SCL:
   "IO BITS".PFR := NOT "SPP";
END_REGION

REGION Network 3: DOOR1 PRESS BIT
   RUNG wire#powerrail
      Contact( "AlwaysTRUE" )
      wire#w1
      { S7_Templates := "SrcType := Real" } GE_Contact(in1 := "PV"."DOOR1 PRESS", in2 := "RETAIN"."SET DOOR1 PRESS HIGH")
      S_Coil( "IO BITS"."DOOR1 PRESS BIT" )
   END_RUNG
   RUNG wire#w1
      { S7_Templates := "SrcType := Real" } LE_Contact(in1 := "PV"."DOOR1 PRESS", in2 := "RETAIN"."SET DOOR1 PRESS LOW")
      R_Coil( "IO BITS"."DOOR1 PRESS BIT" )
   END_RUNG
   // the same network as SCL:
   IF "AlwaysTRUE" AND ("PV"."DOOR1 PRESS" >= "RETAIN"."SET DOOR1 PRESS HIGH") THEN
       "IO BITS"."DOOR1 PRESS BIT" := TRUE;
   END_IF;
   IF "AlwaysTRUE" AND ("PV"."DOOR1 PRESS" <= "RETAIN"."SET DOOR1 PRESS LOW") THEN
       "IO BITS"."DOOR1 PRESS BIT" := FALSE;
   END_IF;
END_REGION

REGION Network 4: DOOR1 VCC BIT
   RUNG wire#powerrail
      Contact( "AlwaysTRUE" )
      { S7_Templates := "SrcType := Real" } LE_Contact(in1 := "PV"."DOOR1 VACCUM", in2 := "RETAIN"."SET DOOR1 VCC")
      Coil( "IO BITS"."DOOR1 VCC BIT" )
   END_RUNG
   // the same network as SCL:
   "IO BITS"."DOOR1 VCC BIT" := "AlwaysTRUE" AND ("PV"."DOOR1 VACCUM" <= "RETAIN"."SET DOOR1 VCC");
END_REGION

REGION Network 5: DOOR2 PRESS BIT
   RUNG wire#powerrail
      Contact( "AlwaysTRUE" )
      wire#w1
      { S7_Templates := "SrcType := Real" } GE_Contact(in1 := "PV"."DOOR2 PRESS", in2 := "RETAIN"."SET DOOR2 PRESS HIGH")
      S_Coil( "IO BITS"."DOOR2 PRESS BIT" )
   END_RUNG
   RUNG wire#w1
      { S7_Templates := "SrcType := Real" } LE_Contact(in1 := "PV"."DOOR2 PRESS", in2 := "RETAIN"."SET DOOR2 PRESS LOW")
      R_Coil( "IO BITS"."DOOR2 PRESS BIT" )
   END_RUNG
   // the same network as SCL:
   IF "AlwaysTRUE" AND ("PV"."DOOR2 PRESS" >= "RETAIN"."SET DOOR2 PRESS HIGH") THEN
       "IO BITS"."DOOR2 PRESS BIT" := TRUE;
   END_IF;
   IF "AlwaysTRUE" AND ("PV"."DOOR2 PRESS" <= "RETAIN"."SET DOOR2 PRESS LOW") THEN
       "IO BITS"."DOOR2 PRESS BIT" := FALSE;
   END_IF;
END_REGION

REGION Network 6: DOOR2 VCC BIT
   RUNG wire#powerrail
      Contact( "AlwaysTRUE" )
      { S7_Templates := "SrcType := Real" } LE_Contact(in1 := "PV"."DOOR2 VACCUM", in2 := "RETAIN"."SET DOOR2 VCC")
      Coil( "IO BITS"."DOOR2 VCC BIT" )
   END_RUNG
   // the same network as SCL:
   "IO BITS"."DOOR2 VCC BIT" := "AlwaysTRUE" AND ("PV"."DOOR2 VACCUM" <= "RETAIN"."SET DOOR2 VCC");
END_REGION

REGION Network 7: JACKET SAFETY BIT
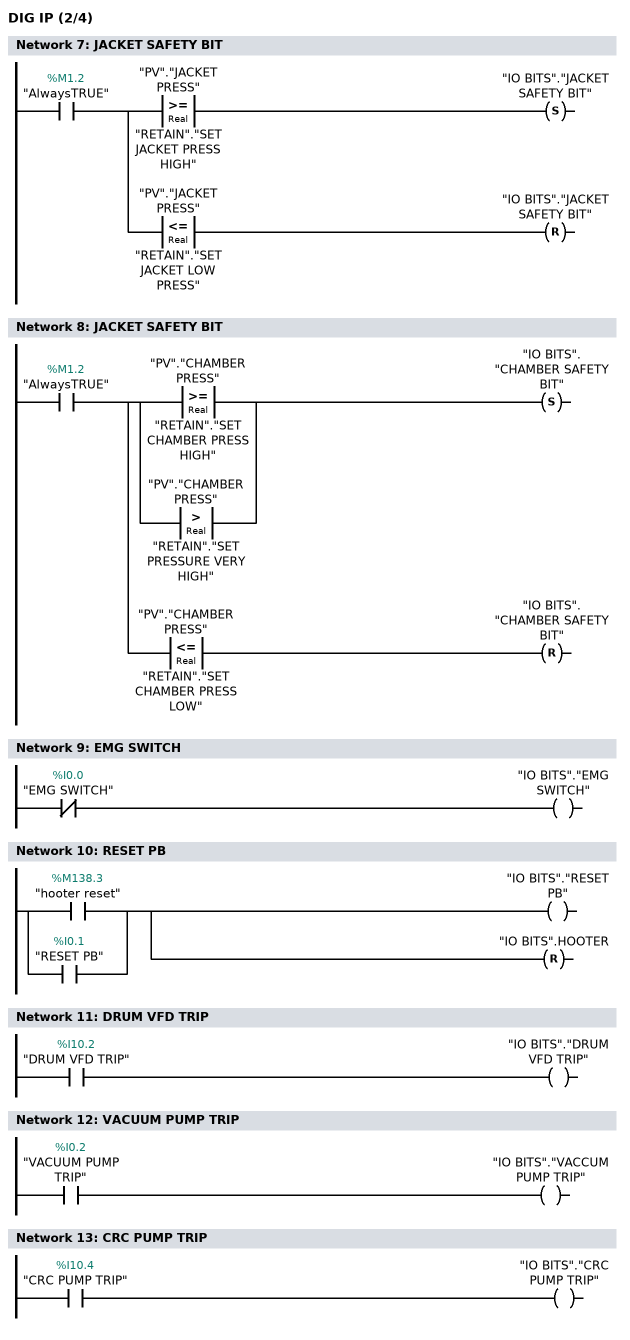
   RUNG wire#powerrail
      Contact( "AlwaysTRUE" )
      wire#w1
      { S7_Templates := "SrcType := Real" } GE_Contact(in1 := "PV"."JACKET PRESS", in2 := "RETAIN"."SET JACKET PRESS HIGH")
      S_Coil( "IO BITS"."JACKET SAFETY BIT" )
   END_RUNG
   RUNG wire#w1
      { S7_Templates := "SrcType := Real" } LE_Contact(in1 := "PV"."JACKET PRESS", in2 := "RETAIN"."SET JACKET LOW PRESS")
      R_Coil( "IO BITS"."JACKET SAFETY BIT" )
   END_RUNG
   // the same network as SCL:
   IF "AlwaysTRUE" AND ("PV"."JACKET PRESS" >= "RETAIN"."SET JACKET PRESS HIGH") THEN
       "IO BITS"."JACKET SAFETY BIT" := TRUE;
   END_IF;
   IF "AlwaysTRUE" AND ("PV"."JACKET PRESS" <= "RETAIN"."SET JACKET LOW PRESS") THEN
       "IO BITS"."JACKET SAFETY BIT" := FALSE;
   END_IF;
END_REGION

REGION Network 8: JACKET SAFETY BIT
   RUNG wire#powerrail
      Contact( "AlwaysTRUE" )
      wire#w1
      { S7_Templates := "SrcType := Real" } GE_Contact(in1 := "PV"."CHAMBER PRESS", in2 := "RETAIN"."SET CHAMBER PRESS HIGH")
      wire#w2
      S_Coil( "IO BITS"."CHAMBER SAFETY BIT" )
   END_RUNG
   RUNG wire#w1
      { S7_Templates := "SrcType := Real" } GT_Contact(in1 := "PV"."CHAMBER PRESS", in2 := "RETAIN"."SET PRESSURE VERY HIGH")
   END_RUNG wire#w2
   RUNG wire#w1
      { S7_Templates := "SrcType := Real" } LE_Contact(in1 := "PV"."CHAMBER PRESS", in2 := "RETAIN"."SET CHAMBER PRESS LOW")
      R_Coil( "IO BITS"."CHAMBER SAFETY BIT" )
   END_RUNG
   // the same network as SCL:
   IF "AlwaysTRUE" AND (("PV"."CHAMBER PRESS" >= "RETAIN"."SET CHAMBER PRESS HIGH") OR ("PV"."CHAMBER PRESS" > "RETAIN"."SET PRESSURE VERY HIGH")) THEN
       "IO BITS"."CHAMBER SAFETY BIT" := TRUE;
   END_IF;
   IF "AlwaysTRUE" AND ("PV"."CHAMBER PRESS" <= "RETAIN"."SET CHAMBER PRESS LOW") THEN
       "IO BITS"."CHAMBER SAFETY BIT" := FALSE;
   END_IF;
END_REGION

REGION Network 9: EMG SWITCH
   RUNG wire#powerrail
      I_Contact( "EMG SWITCH" )
      Coil( "IO BITS"."EMG SWITCH" )
   END_RUNG
   // the same network as SCL:
   "IO BITS"."EMG SWITCH" := NOT "EMG SWITCH";
END_REGION

REGION Network 10: RESET PB
   RUNG wire#powerrail
      Contact( "hooter reset" )
      wire#w1
      Coil( "IO BITS"."RESET PB" )
   END_RUNG
   RUNG wire#powerrail
      Contact( "RESET PB" )
   END_RUNG wire#w1
   RUNG wire#w1
      R_Coil( "IO BITS".HOOTER )
   END_RUNG
   // the same network as SCL:
   "IO BITS"."RESET PB" := "hooter reset" OR "RESET PB";
   IF "IO BITS"."RESET PB" THEN "IO BITS".HOOTER := FALSE; END_IF;
END_REGION

REGION Network 11: DRUM VFD TRIP
   RUNG wire#powerrail
      Contact( "DRUM VFD TRIP" )
      Coil( "IO BITS"."DRUM VFD TRIP" )
   END_RUNG
   // the same network as SCL:
   "IO BITS"."DRUM VFD TRIP" := "DRUM VFD TRIP";
END_REGION

REGION Network 12: VACUUM PUMP TRIP
   RUNG wire#powerrail
      Contact( "VACUUM PUMP TRIP" )
      Coil( "IO BITS"."VACCUM PUMP TRIP" )
   END_RUNG
   // the same network as SCL:
   "IO BITS"."VACCUM PUMP TRIP" := "VACUUM PUMP TRIP";
END_REGION

REGION Network 13: CRC PUMP TRIP
   RUNG wire#powerrail
      Contact( "CRC PUMP TRIP" )
      Coil( "IO BITS"."CRC PUMP TRIP" )
   END_RUNG
   // the same network as SCL:
   "IO BITS"."CRC PUMP TRIP" := "CRC PUMP TRIP";
END_REGION

REGION Network 14: DOOR1 OPEN LMT
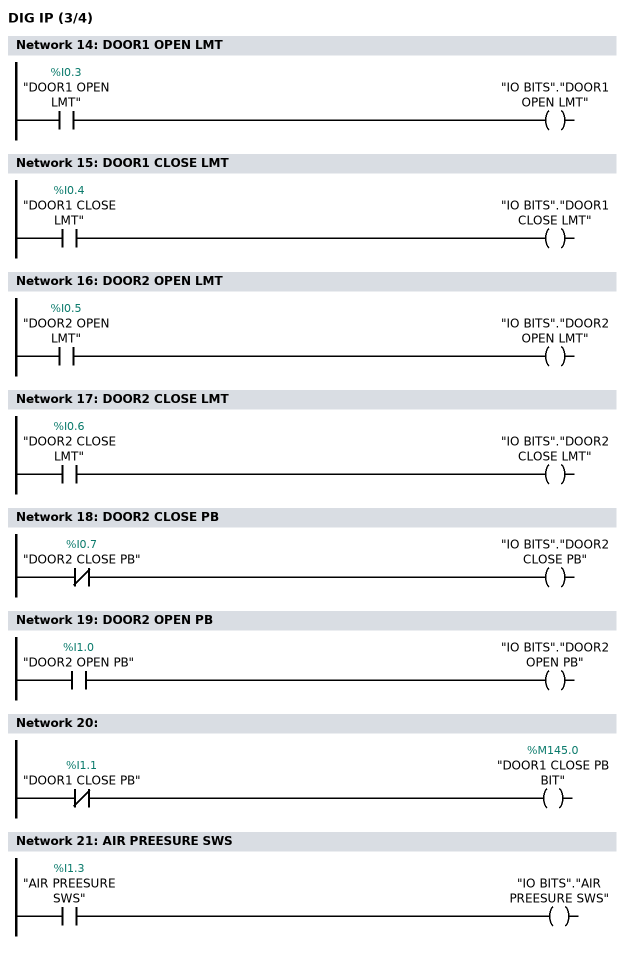
   RUNG wire#powerrail
      Contact( "DOOR1 OPEN LMT" )
      Coil( "IO BITS"."DOOR1 OPEN LMT" )
   END_RUNG
   // the same network as SCL:
   "IO BITS"."DOOR1 OPEN LMT" := "DOOR1 OPEN LMT";
END_REGION

REGION Network 15: DOOR1 CLOSE LMT
   RUNG wire#powerrail
      Contact( "DOOR1 CLOSE LMT" )
      Coil( "IO BITS"."DOOR1 CLOSE LMT" )
   END_RUNG
   // the same network as SCL:
   "IO BITS"."DOOR1 CLOSE LMT" := "DOOR1 CLOSE LMT";
END_REGION

REGION Network 16: DOOR2 OPEN LMT
   RUNG wire#powerrail
      Contact( "DOOR2 OPEN LMT" )
      Coil( "IO BITS"."DOOR2 OPEN LMT" )
   END_RUNG
   // the same network as SCL:
   "IO BITS"."DOOR2 OPEN LMT" := "DOOR2 OPEN LMT";
END_REGION

REGION Network 17: DOOR2 CLOSE LMT
   RUNG wire#powerrail
      Contact( "DOOR2 CLOSE LMT" )
      Coil( "IO BITS"."DOOR2 CLOSE LMT" )
   END_RUNG
   // the same network as SCL:
   "IO BITS"."DOOR2 CLOSE LMT" := "DOOR2 CLOSE LMT";
END_REGION

REGION Network 18: DOOR2 CLOSE PB
   RUNG wire#powerrail
      I_Contact( "DOOR2 CLOSE PB" )
      Coil( "IO BITS"."DOOR2 CLOSE PB" )
   END_RUNG
   // the same network as SCL:
   "IO BITS"."DOOR2 CLOSE PB" := NOT "DOOR2 CLOSE PB";
END_REGION

REGION Network 19: DOOR2 OPEN PB
   RUNG wire#powerrail
      Contact( "DOOR2 OPEN PB" )
      Coil( "IO BITS"."DOOR2 OPEN PB" )
   END_RUNG
   // the same network as SCL:
   "IO BITS"."DOOR2 OPEN PB" := "DOOR2 OPEN PB";
END_REGION

REGION Network 20
   RUNG wire#powerrail
      I_Contact( "DOOR1 CLOSE PB" )
      Coil( "DOOR1 CLOSE PB BIT" )
   END_RUNG
   // the same network as SCL:
   "DOOR1 CLOSE PB BIT" := NOT "DOOR1 CLOSE PB";
END_REGION

REGION Network 21: AIR PREESURE SWS
   RUNG wire#powerrail
      Contact( "AIR PREESURE SWS" )
      Coil( "IO BITS"."AIR PREESURE SWS" )
   END_RUNG
   // the same network as SCL:
   "IO BITS"."AIR PREESURE SWS" := "AIR PREESURE SWS";
END_REGION

REGION Network 22
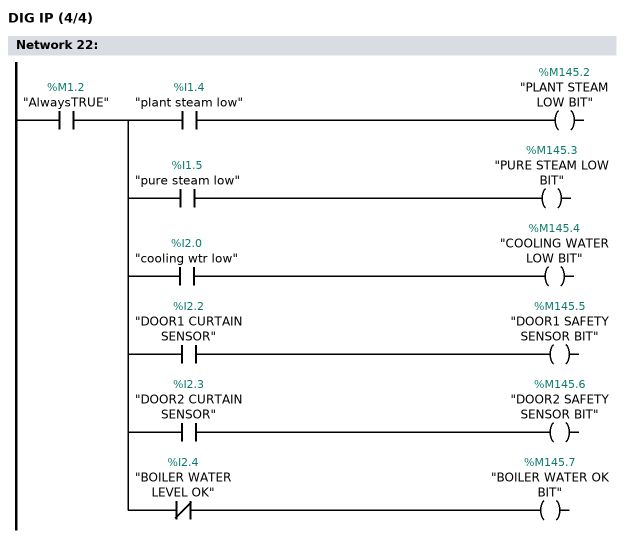
   RUNG wire#powerrail
      Contact( "AlwaysTRUE" )
      wire#w1
      Contact( "plant steam low" )
      Coil( "PLANT STEAM LOW BIT" )
   END_RUNG
   RUNG wire#w1
      Contact( "pure steam low" )
      Coil( "PURE STEAM LOW BIT" )
   END_RUNG
   RUNG wire#w1
      Contact( "cooling wtr low" )
      Coil( "COOLING WATER LOW BIT" )
   END_RUNG
   RUNG wire#w1
      Contact( "DOOR1 CURTAIN SENSOR" )
      Coil( "DOOR1 SAFETY SENSOR BIT" )
   END_RUNG
   RUNG wire#w1
      Contact( "DOOR2 CURTAIN SENSOR" )
      Coil( "DOOR2 SAFETY SENSOR BIT" )
   END_RUNG
   RUNG wire#w1
      I_Contact( "BOILER WATER LEVEL OK" )
      Coil( "BOILER WATER OK BIT" )
   END_RUNG
   // the same network as SCL:
   "PLANT STEAM LOW BIT" := "AlwaysTRUE" AND "plant steam low";
   "PURE STEAM LOW BIT" := "AlwaysTRUE" AND "pure steam low";
   "COOLING WATER LOW BIT" := "AlwaysTRUE" AND "cooling wtr low";
   "DOOR1 SAFETY SENSOR BIT" := "AlwaysTRUE" AND "DOOR1 CURTAIN SENSOR";
   "DOOR2 SAFETY SENSOR BIT" := "AlwaysTRUE" AND "DOOR2 CURTAIN SENSOR";
   "BOILER WATER OK BIT" := "AlwaysTRUE" AND NOT "BOILER WATER LEVEL OK";
END_REGION
END_FUNCTION

FUNCTION "STANDARD" : Void   // FC13, LAD
{ S7_Optimized_Access := 'TRUE' }
// stored: SetENOAutomatically false
   VAR_TEMP
      "std temp3 hyst" : Real;
   END_VAR
   VAR_TEMP   // added for the SCL form of the ladder/FBD networks
      _w1 : Bool;
      _w2 : Bool;
      _w3 : Bool;
      _w4 : Bool;
   END_VAR
BEGIN

REGION Network 1
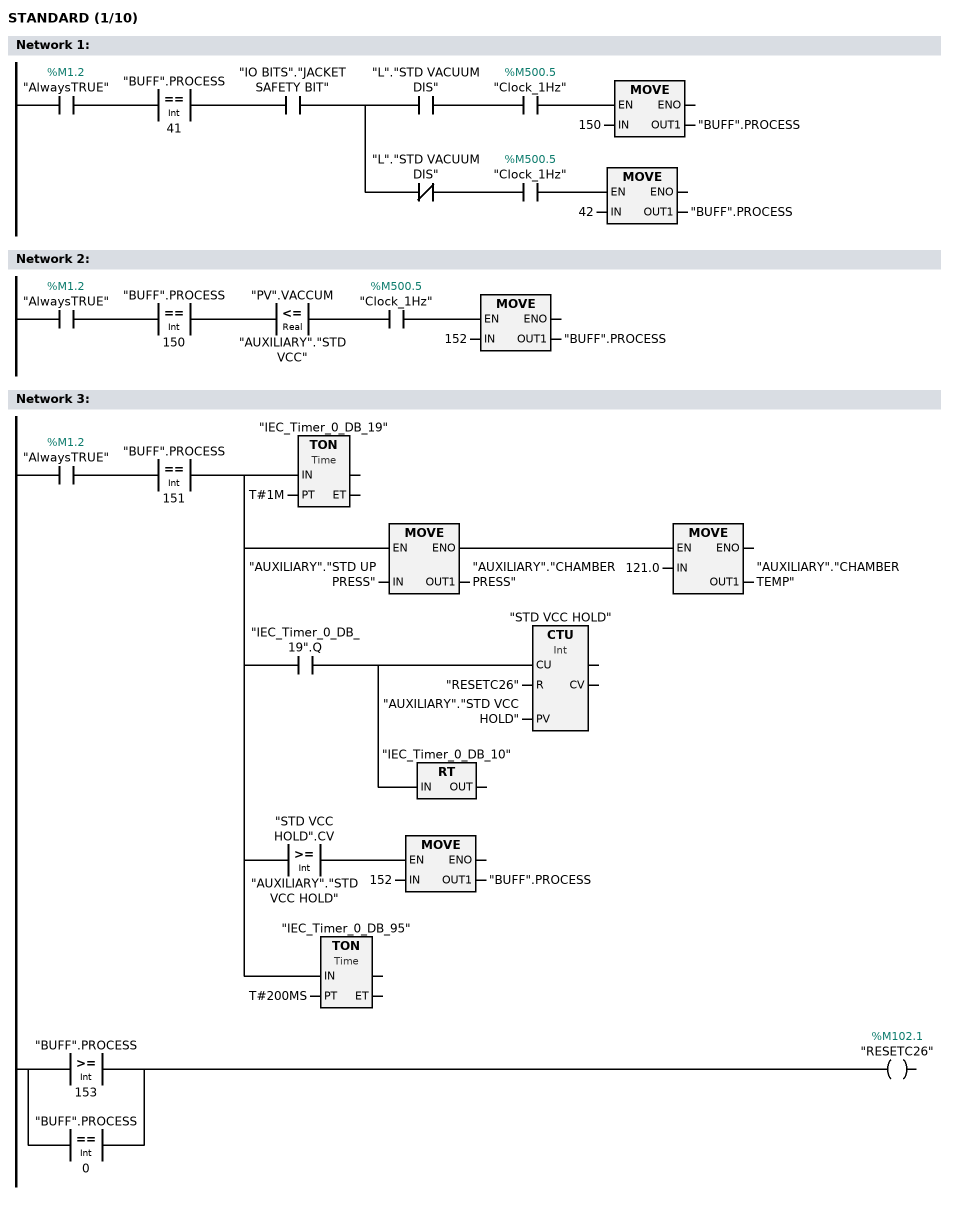
   RUNG wire#powerrail
      Contact( "AlwaysTRUE" )
      { S7_Templates := "SrcType := Int" } EQ_Contact(in1 := "BUFF".PROCESS, in2 := 41)
      Contact( "IO BITS"."JACKET SAFETY BIT" )
      wire#w1
      Contact( "L"."STD VACUUM DIS" )
      Contact( "Clock_1Hz" )
      Move(in := 150, out1 => "BUFF".PROCESS)
   END_RUNG
   RUNG wire#w1
      I_Contact( "L"."STD VACUUM DIS" )
      Contact( "Clock_1Hz" )
      Move(in := 42, out1 => "BUFF".PROCESS)
   END_RUNG
   // the same network as SCL:
   #_w1 := "AlwaysTRUE" AND ("BUFF".PROCESS = 41) AND "IO BITS"."JACKET SAFETY BIT";
   IF #_w1 AND "L"."STD VACUUM DIS" AND "Clock_1Hz" THEN "BUFF".PROCESS := 150; END_IF;
   IF #_w1 AND NOT "L"."STD VACUUM DIS" AND "Clock_1Hz" THEN "BUFF".PROCESS := 42; END_IF;
END_REGION

REGION Network 2
   RUNG wire#powerrail
      Contact( "AlwaysTRUE" )
      { S7_Templates := "SrcType := Int" } EQ_Contact(in1 := "BUFF".PROCESS, in2 := 150)
      { S7_Templates := "SrcType := Real" } LE_Contact(in1 := "PV".VACCUM, in2 := "AUXILIARY"."STD VCC")
      Contact( "Clock_1Hz" )
      Move(in := 152, out1 => "BUFF".PROCESS)
   END_RUNG
   // the same network as SCL:
   IF "AlwaysTRUE" AND ("BUFF".PROCESS = 150) AND ("PV".VACCUM <= "AUXILIARY"."STD VCC") AND "Clock_1Hz" THEN
       "BUFF".PROCESS := 152;
   END_IF;
END_REGION

REGION Network 3
   RUNG wire#powerrail
      Contact( "AlwaysTRUE" )
      { S7_Templates := "SrcType := Int" } EQ_Contact(in1 := "BUFF".PROCESS, in2 := 151)
      wire#w1
      { S7_Templates := "time_type := Time" } "IEC_Timer_0_DB_19".TON(pt := T#1M, et =>)
   END_RUNG
   RUNG wire#w1
      Move(in := "AUXILIARY"."STD UP PRESS", out1 => "AUXILIARY"."CHAMBER PRESS")
      Move(in := 121.0, out1 => "AUXILIARY"."CHAMBER TEMP")
   END_RUNG
   RUNG wire#w1
      Contact( "IEC_Timer_0_DB_19".Q )
      wire#w2
      { S7_Templates := "value_type := Int" } "STD VCC HOLD".CTU(r := "RESETC26", pv := "AUXILIARY"."STD VCC HOLD", cv =>)
   END_RUNG
   RUNG wire#w2
      RT_Coil( "IEC_Timer_0_DB_10" )
   END_RUNG
   RUNG wire#w1
      { S7_Templates := "SrcType := Int" } GE_Contact(in1 := "STD VCC HOLD".CV, in2 := "AUXILIARY"."STD VCC HOLD")
      Move(in := 152, out1 => "BUFF".PROCESS)
   END_RUNG
   RUNG wire#w1
      { S7_Templates := "time_type := Time" } "IEC_Timer_0_DB_95".TON(pt := T#200MS, et =>)
   END_RUNG
   RUNG wire#powerrail
      { S7_Templates := "SrcType := Int" } GE_Contact(in1 := "BUFF".PROCESS, in2 := 153)
      wire#w3
      Coil( "RESETC26" )
   END_RUNG
   RUNG wire#powerrail
      { S7_Templates := "SrcType := Int" } EQ_Contact(in1 := "BUFF".PROCESS, in2 := 0)
   END_RUNG wire#w3
   // the same network as SCL:
   #_w1 := "AlwaysTRUE" AND ("BUFF".PROCESS = 151);
   "IEC_Timer_0_DB_19".TON(IN := #_w1, PT := T#1M);
   IF #_w1 THEN
       "AUXILIARY"."CHAMBER PRESS" := "AUXILIARY"."STD UP PRESS";
       "AUXILIARY"."CHAMBER TEMP" := 121.0;
   END_IF;
   #_w2 := #_w1 AND "IEC_Timer_0_DB_19".Q;
   "STD VCC HOLD".CTU(CU := #_w2, R := "RESETC26", PV := "AUXILIARY"."STD VCC HOLD");
   IF #_w2 THEN RESET_TIMER("IEC_Timer_0_DB_10"); END_IF;
   IF #_w1 AND ("STD VCC HOLD".CV >= "AUXILIARY"."STD VCC HOLD") THEN "BUFF".PROCESS := 152; END_IF;
   "IEC_Timer_0_DB_95".TON(IN := #_w1, PT := T#200MS);
   "RESETC26" := ("BUFF".PROCESS >= 153) OR ("BUFF".PROCESS = 0);
END_REGION

REGION Network 4
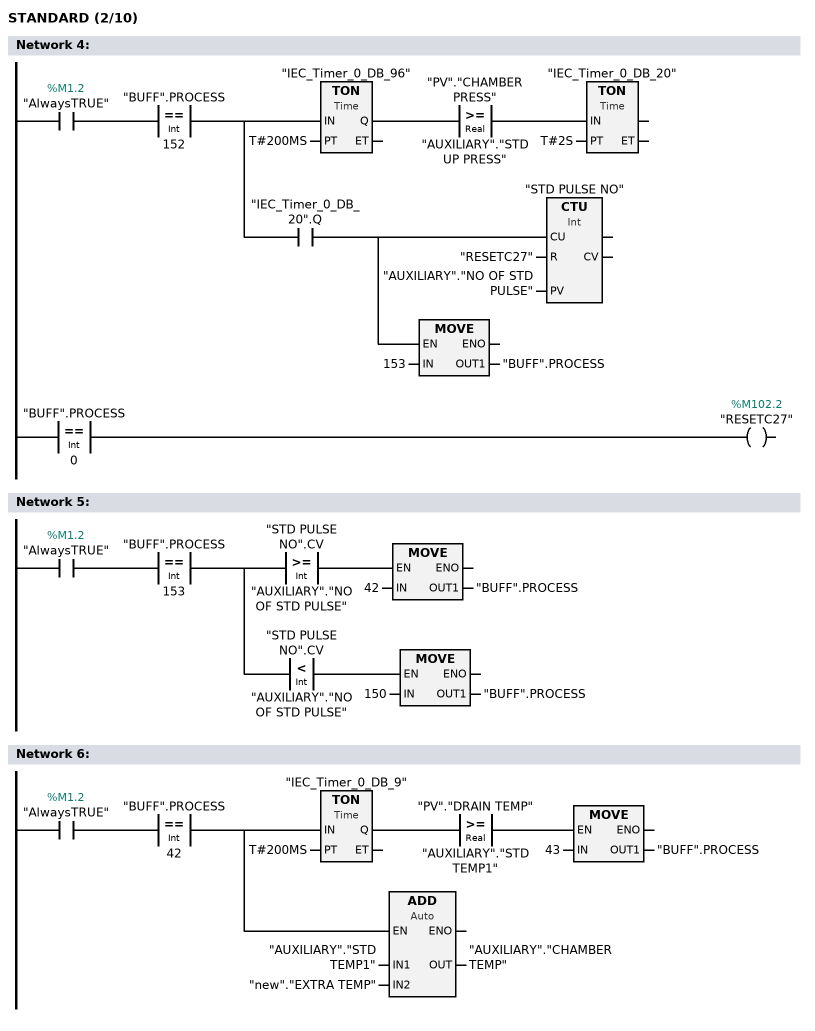
   RUNG wire#powerrail
      Contact( "AlwaysTRUE" )
      { S7_Templates := "SrcType := Int" } EQ_Contact(in1 := "BUFF".PROCESS, in2 := 152)
      wire#w1
      { S7_Templates := "time_type := Time" } "IEC_Timer_0_DB_96".TON(pt := T#200MS, et =>)
      { S7_Templates := "SrcType := Real" } GE_Contact(in1 := "PV"."CHAMBER PRESS", in2 := "AUXILIARY"."STD UP PRESS")
      { S7_Templates := "time_type := Time" } "IEC_Timer_0_DB_20".TON(pt := T#2S, et =>)
   END_RUNG
   RUNG wire#w1
      Contact( "IEC_Timer_0_DB_20".Q )
      wire#w2
      { S7_Templates := "value_type := Int" } "STD PULSE NO".CTU(r := "RESETC27", pv := "AUXILIARY"."NO OF STD PULSE", cv =>)
   END_RUNG
   RUNG wire#w2
      Move(in := 153, out1 => "BUFF".PROCESS)
   END_RUNG
   RUNG wire#powerrail
      { S7_Templates := "SrcType := Int" } EQ_Contact(in1 := "BUFF".PROCESS, in2 := 0)
      Coil( "RESETC27" )
   END_RUNG
   // the same network as SCL:
   #_w1 := "AlwaysTRUE" AND ("BUFF".PROCESS = 152);
   "IEC_Timer_0_DB_96".TON(IN := #_w1, PT := T#200MS);
   "IEC_Timer_0_DB_20".TON(IN := "IEC_Timer_0_DB_96".Q AND ("PV"."CHAMBER PRESS" >= "AUXILIARY"."STD UP PRESS"),
                           PT := T#2S);
   #_w2 := #_w1 AND "IEC_Timer_0_DB_20".Q;
   "STD PULSE NO".CTU(CU := #_w2, R := "RESETC27", PV := "AUXILIARY"."NO OF STD PULSE");
   IF #_w2 THEN "BUFF".PROCESS := 153; END_IF;
   "RESETC27" := "BUFF".PROCESS = 0;
END_REGION

REGION Network 5
   RUNG wire#powerrail
      Contact( "AlwaysTRUE" )
      { S7_Templates := "SrcType := Int" } EQ_Contact(in1 := "BUFF".PROCESS, in2 := 153)
      wire#w1
      { S7_Templates := "SrcType := Int" } GE_Contact(in1 := "STD PULSE NO".CV, in2 := "AUXILIARY"."NO OF STD PULSE")
      Move(in := 42, out1 => "BUFF".PROCESS)
   END_RUNG
   RUNG wire#w1
      { S7_Templates := "SrcType := Int" } LT_Contact(in1 := "STD PULSE NO".CV, in2 := "AUXILIARY"."NO OF STD PULSE")
      Move(in := 150, out1 => "BUFF".PROCESS)
   END_RUNG
   // the same network as SCL:
   #_w1 := "AlwaysTRUE" AND ("BUFF".PROCESS = 153);
   IF #_w1 AND ("STD PULSE NO".CV >= "AUXILIARY"."NO OF STD PULSE") THEN "BUFF".PROCESS := 42; END_IF;
   IF #_w1 AND ("STD PULSE NO".CV < "AUXILIARY"."NO OF STD PULSE") THEN "BUFF".PROCESS := 150; END_IF;
END_REGION

REGION Network 6
   RUNG wire#powerrail
      Contact( "AlwaysTRUE" )
      { S7_Templates := "SrcType := Int" } EQ_Contact(in1 := "BUFF".PROCESS, in2 := 42)
      wire#w1
      { S7_Templates := "time_type := Time" } "IEC_Timer_0_DB_9".TON(pt := T#200MS, et =>)
      { S7_Templates := "SrcType := Real" } GE_Contact(in1 := "PV"."DRAIN TEMP", in2 := "AUXILIARY"."STD TEMP1")
      Move(in := 43, out1 => "BUFF".PROCESS)
   END_RUNG
   RUNG wire#w1
      Add(in1 := "AUXILIARY"."STD TEMP1", in2 := "new"."EXTRA TEMP", out => "AUXILIARY"."CHAMBER TEMP")
   END_RUNG
   // the same network as SCL:
   #_w1 := "AlwaysTRUE" AND ("BUFF".PROCESS = 42);
   "IEC_Timer_0_DB_9".TON(IN := #_w1, PT := T#200MS);
   IF "IEC_Timer_0_DB_9".Q AND ("PV"."DRAIN TEMP" >= "AUXILIARY"."STD TEMP1") THEN
       "BUFF".PROCESS := 43;
   END_IF;
   IF #_w1 THEN "AUXILIARY"."CHAMBER TEMP" := "AUXILIARY"."STD TEMP1" + "new"."EXTRA TEMP"; END_IF;
END_REGION

REGION Network 7
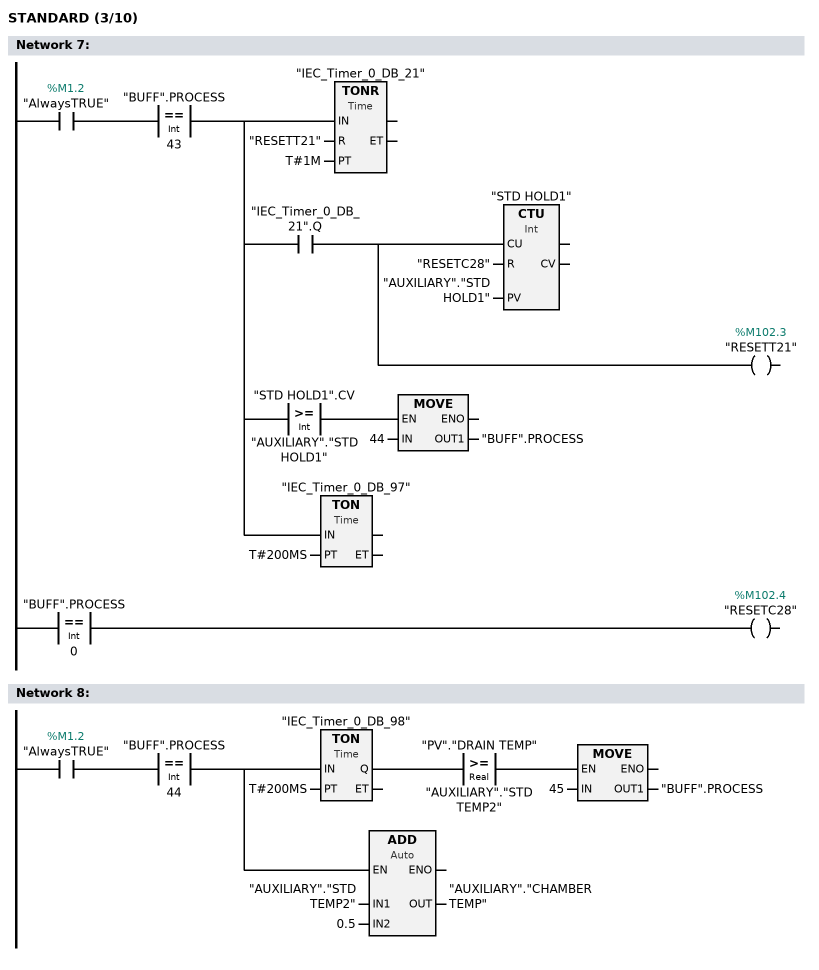
   RUNG wire#powerrail
      Contact( "AlwaysTRUE" )
      { S7_Templates := "SrcType := Int" } EQ_Contact(in1 := "BUFF".PROCESS, in2 := 43)
      wire#w1
      { S7_Templates := "time_type := Time" } "IEC_Timer_0_DB_21".TONR(r := "RESETT21", pt := T#1M, et =>)
   END_RUNG
   RUNG wire#w1
      Contact( "IEC_Timer_0_DB_21".Q )
      wire#w2
      { S7_Templates := "value_type := Int" } "STD HOLD1".CTU(r := "RESETC28", pv := "AUXILIARY"."STD HOLD1", cv =>)
   END_RUNG
   RUNG wire#w2
      Coil( "RESETT21" )
   END_RUNG
   RUNG wire#w1
      { S7_Templates := "SrcType := Int" } GE_Contact(in1 := "STD HOLD1".CV, in2 := "AUXILIARY"."STD HOLD1")
      Move(in := 44, out1 => "BUFF".PROCESS)
   END_RUNG
   RUNG wire#w1
      { S7_Templates := "time_type := Time" } "IEC_Timer_0_DB_97".TON(pt := T#200MS, et =>)
   END_RUNG
   RUNG wire#powerrail
      { S7_Templates := "SrcType := Int" } EQ_Contact(in1 := "BUFF".PROCESS, in2 := 0)
      Coil( "RESETC28" )
   END_RUNG
   // the same network as SCL:
   #_w1 := "AlwaysTRUE" AND ("BUFF".PROCESS = 43);
   "IEC_Timer_0_DB_21".TONR(IN := #_w1, R := "RESETT21", PT := T#1M);
   #_w2 := #_w1 AND "IEC_Timer_0_DB_21".Q;
   "STD HOLD1".CTU(CU := #_w2, R := "RESETC28", PV := "AUXILIARY"."STD HOLD1");
   "RESETT21" := #_w2;
   IF #_w1 AND ("STD HOLD1".CV >= "AUXILIARY"."STD HOLD1") THEN "BUFF".PROCESS := 44; END_IF;
   "IEC_Timer_0_DB_97".TON(IN := #_w1, PT := T#200MS);
   "RESETC28" := "BUFF".PROCESS = 0;
END_REGION

REGION Network 8
   RUNG wire#powerrail
      Contact( "AlwaysTRUE" )
      { S7_Templates := "SrcType := Int" } EQ_Contact(in1 := "BUFF".PROCESS, in2 := 44)
      wire#w1
      { S7_Templates := "time_type := Time" } "IEC_Timer_0_DB_98".TON(pt := T#200MS, et =>)
      { S7_Templates := "SrcType := Real" } GE_Contact(in1 := "PV"."DRAIN TEMP", in2 := "AUXILIARY"."STD TEMP2")
      Move(in := 45, out1 => "BUFF".PROCESS)
   END_RUNG
   RUNG wire#w1
      Add(in1 := "AUXILIARY"."STD TEMP2", in2 := 0.5, out => "AUXILIARY"."CHAMBER TEMP")
   END_RUNG
   // the same network as SCL:
   #_w1 := "AlwaysTRUE" AND ("BUFF".PROCESS = 44);
   "IEC_Timer_0_DB_98".TON(IN := #_w1, PT := T#200MS);
   IF "IEC_Timer_0_DB_98".Q AND ("PV"."DRAIN TEMP" >= "AUXILIARY"."STD TEMP2") THEN
       "BUFF".PROCESS := 45;
   END_IF;
   IF #_w1 THEN "AUXILIARY"."CHAMBER TEMP" := "AUXILIARY"."STD TEMP2" + 0.5; END_IF;
END_REGION

REGION Network 9
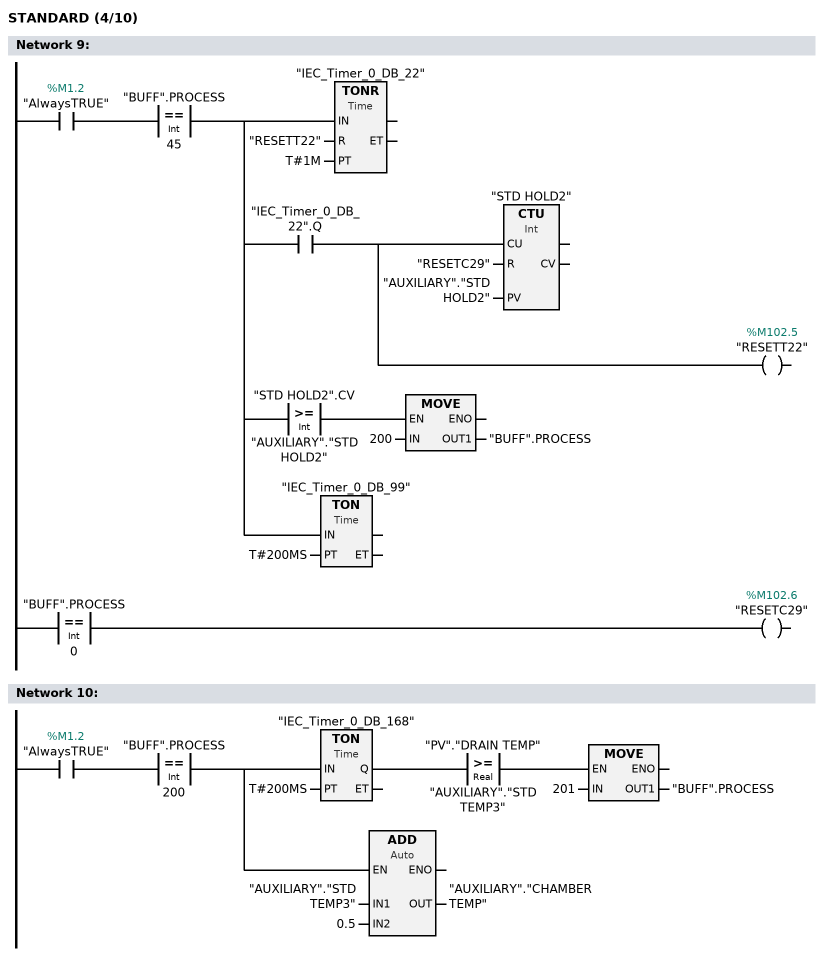
   RUNG wire#powerrail
      Contact( "AlwaysTRUE" )
      { S7_Templates := "SrcType := Int" } EQ_Contact(in1 := "BUFF".PROCESS, in2 := 45)
      wire#w1
      { S7_Templates := "time_type := Time" } "IEC_Timer_0_DB_22".TONR(r := "RESETT22", pt := T#1M, et =>)
   END_RUNG
   RUNG wire#w1
      Contact( "IEC_Timer_0_DB_22".Q )
      wire#w2
      { S7_Templates := "value_type := Int" } "STD HOLD2".CTU(r := "RESETC29", pv := "AUXILIARY"."STD HOLD2", cv =>)
   END_RUNG
   RUNG wire#w2
      Coil( "RESETT22" )
   END_RUNG
   RUNG wire#w1
      { S7_Templates := "SrcType := Int" } GE_Contact(in1 := "STD HOLD2".CV, in2 := "AUXILIARY"."STD HOLD2")
      Move(in := 200, out1 => "BUFF".PROCESS)
   END_RUNG
   RUNG wire#w1
      { S7_Templates := "time_type := Time" } "IEC_Timer_0_DB_99".TON(pt := T#200MS, et =>)
   END_RUNG
   RUNG wire#powerrail
      { S7_Templates := "SrcType := Int" } EQ_Contact(in1 := "BUFF".PROCESS, in2 := 0)
      Coil( "RESETC29" )
   END_RUNG
   // the same network as SCL:
   #_w1 := "AlwaysTRUE" AND ("BUFF".PROCESS = 45);
   "IEC_Timer_0_DB_22".TONR(IN := #_w1, R := "RESETT22", PT := T#1M);
   #_w2 := #_w1 AND "IEC_Timer_0_DB_22".Q;
   "STD HOLD2".CTU(CU := #_w2, R := "RESETC29", PV := "AUXILIARY"."STD HOLD2");
   "RESETT22" := #_w2;
   IF #_w1 AND ("STD HOLD2".CV >= "AUXILIARY"."STD HOLD2") THEN "BUFF".PROCESS := 200; END_IF;
   "IEC_Timer_0_DB_99".TON(IN := #_w1, PT := T#200MS);
   "RESETC29" := "BUFF".PROCESS = 0;
END_REGION

REGION Network 10
   RUNG wire#powerrail
      Contact( "AlwaysTRUE" )
      { S7_Templates := "SrcType := Int" } EQ_Contact(in1 := "BUFF".PROCESS, in2 := 200)
      wire#w1
      { S7_Templates := "time_type := Time" } "IEC_Timer_0_DB_168".TON(pt := T#200MS, et =>)
      { S7_Templates := "SrcType := Real" } GE_Contact(in1 := "PV"."DRAIN TEMP", in2 := "AUXILIARY"."STD TEMP3")
      Move(in := 201, out1 => "BUFF".PROCESS)
   END_RUNG
   RUNG wire#w1
      Add(in1 := "AUXILIARY"."STD TEMP3", in2 := 0.5, out => "AUXILIARY"."CHAMBER TEMP")
   END_RUNG
   // the same network as SCL:
   #_w1 := "AlwaysTRUE" AND ("BUFF".PROCESS = 200);
   "IEC_Timer_0_DB_168".TON(IN := #_w1, PT := T#200MS);
   IF "IEC_Timer_0_DB_168".Q AND ("PV"."DRAIN TEMP" >= "AUXILIARY"."STD TEMP3") THEN
       "BUFF".PROCESS := 201;
   END_IF;
   IF #_w1 THEN "AUXILIARY"."CHAMBER TEMP" := "AUXILIARY"."STD TEMP3" + 0.5; END_IF;
END_REGION

REGION Network 11
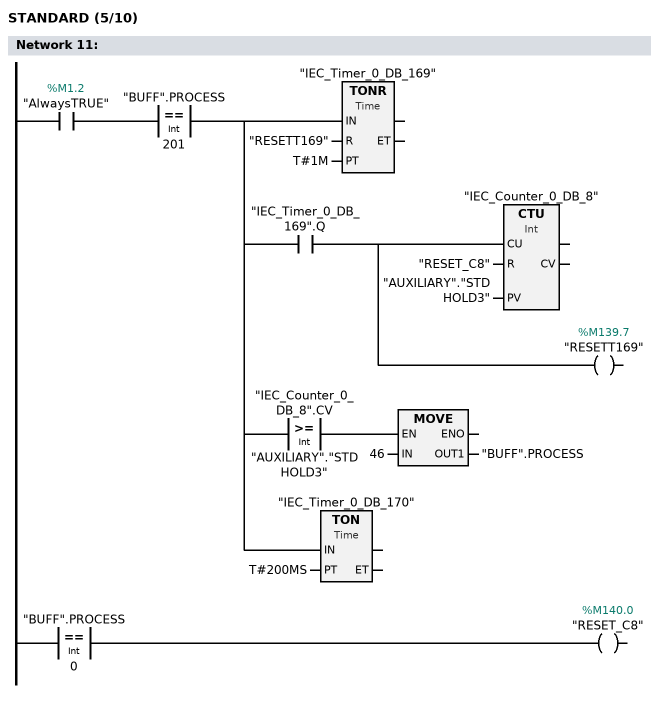
   RUNG wire#powerrail
      Contact( "AlwaysTRUE" )
      { S7_Templates := "SrcType := Int" } EQ_Contact(in1 := "BUFF".PROCESS, in2 := 201)
      wire#w1
      { S7_Templates := "time_type := Time" } "IEC_Timer_0_DB_169".TONR(r := "RESETT169", pt := T#1M, et =>)
   END_RUNG
   RUNG wire#w1
      Contact( "IEC_Timer_0_DB_169".Q )
      wire#w2
      { S7_Templates := "value_type := Int" } "IEC_Counter_0_DB_8".CTU(r := "RESET_C8", pv := "AUXILIARY"."STD HOLD3", cv =>)
   END_RUNG
   RUNG wire#w2
      Coil( "RESETT169" )
   END_RUNG
   RUNG wire#w1
      { S7_Templates := "SrcType := Int" } GE_Contact(in1 := "IEC_Counter_0_DB_8".CV, in2 := "AUXILIARY"."STD HOLD3")
      Move(in := 46, out1 => "BUFF".PROCESS)
   END_RUNG
   RUNG wire#w1
      { S7_Templates := "time_type := Time" } "IEC_Timer_0_DB_170".TON(pt := T#200MS, et =>)
   END_RUNG
   RUNG wire#powerrail
      { S7_Templates := "SrcType := Int" } EQ_Contact(in1 := "BUFF".PROCESS, in2 := 0)
      Coil( "RESET_C8" )
   END_RUNG
   // the same network as SCL:
   #_w1 := "AlwaysTRUE" AND ("BUFF".PROCESS = 201);
   "IEC_Timer_0_DB_169".TONR(IN := #_w1, R := "RESETT169", PT := T#1M);
   #_w2 := #_w1 AND "IEC_Timer_0_DB_169".Q;
   "IEC_Counter_0_DB_8".CTU(CU := #_w2, R := "RESET_C8", PV := "AUXILIARY"."STD HOLD3");
   "RESETT169" := #_w2;
   IF #_w1 AND ("IEC_Counter_0_DB_8".CV >= "AUXILIARY"."STD HOLD3") THEN "BUFF".PROCESS := 46; END_IF;
   "IEC_Timer_0_DB_170".TON(IN := #_w1, PT := T#200MS);
   "RESET_C8" := "BUFF".PROCESS = 0;
END_REGION

REGION Network 12
